LIN {X 0,Y 364.945,Z 184.267,A -85,B 0,C 180,E1 -13027.295,E2 -13027.295} C_VEL
LIN {X 0,Y 368.82,Z 205.112,A -85,B 0,C 180,E1 -13028.057,E2 -13028.057} C_VEL
LIN {X 0,Y 371.05,Z 221.35,A -85,B 0,C 180,E1 -13028.583,E2 -13028.583} C_VEL
LIN {X 0,Y 369.557,Z 293.97,A -85,B 0,C 180,E1 -13030.126,E2 -13030.126} C_VEL
LIN {X 0,Y 368.772,Z 307.522,A -85,B 0,C 180,E1 -13030.626,E2 -13030.626} C_VEL
LIN {X 0,Y 367.784,Z 320.407,A -85,B 0,C 180,E1 -13031.332,E2 -13031.332} C_VEL
LIN {X 0,Y 366.724,Z 331.401,A -85,B 0,C 180,E1 -13032.143,E2 -13032.143} C_VEL
LIN {X 0,Y 365.474,Z 342.946,A -85,B 0,C 180,E1 -13033.234,E2 -13033.234} C_VEL
LIN {X 0,Y 364.338,Z 353.389,A -85,B 0,C 180,E1 -13034.475,E2 -13034.475} C_VEL
LIN {X 0,Y 363.355,Z 361.959,A -85,B 0,C 180,E1 -13035.722,E2 -13035.722} C_VEL
LIN {X 0,Y 362.336,Z 371.27,A -85,B 0,C 180,E1 -13037.395,E2 -13037.395} C_VEL
LIN {X 0,Y 361.44,Z 378.781,A -85,B 0,C 180,E1 -13039.071,E2 -13039.071} C_VEL
LIN {X 0,Y 360.832,Z 385.726,A -85,B 0,C 180,E1 -13041.035,E2 -13041.035} C_VEL
LIN {X 0,Y 360.514,Z 390.327,A -85,B 0,C 180,E1 -13042.72,E2 -13042.72} C_VEL
LIN {X 0,Y 360.354,Z 393.835,A -85,B 0,C 180,E1 -13044.403,E2 -13044.403} C_VEL
LIN {X 0,Y 360.362,Z 395.591,A -85,B 0,C 180,E1 -13045.525,E2 -13045.525} C_VEL
LIN {X 0,Y 360.327,Z 396.936,A -85,B 0,C 180,E1 -13046.645,E2 -13046.645} C_VEL
LIN {X 0,Y 360.353,Z 397.882,A -85,B 0,C 180,E1 -13047.764,E2 -13047.764} C_VEL
LIN {X 0,Y 360.457,Z 398.389,A -85,B 0,C 180,E1 -13048.882,E2 -13048.882} C_VEL
LIN {X 0,Y 360.482,Z 398.479,A -85,B 0,C 180,E1 -13049.999,E2 -13049.999} C_VEL
LIN {X 0,Y 360.459,Z 398.172,A -85,B 0,C 180,E1 -13051.117,E2 -13051.117} C_VEL
LIN {X 0,Y 360.372,Z 397.464,A -85,B 0,C 180,E1 -13052.235,E2 -13052.235} C_VEL
LIN {X 0,Y 360.332,Z 396.308,A -85,B 0,C 180,E1 -13053.354,E2 -13053.354} C_VEL
LIN {X 0,Y 360.343,Z 393.784,A -85,B 0,C 180,E1 -13055.034,E2 -13055.034} C_VEL
LIN {X 0,Y 360.486,Z 390.224,A -85,B 0,C 180,E1 -13056.717,E2 -13056.717} C_VEL
LIN {X 0,Y 360.691,Z 385.523,A -85,B 0,C 180,E1 -13058.402,E2 -13058.402} C_VEL
LIN {X 0,Y 361.168,Z 378.413,A -85,B 0,C 180,E1 -13060.369,E2 -13060.369} C_VEL
LIN {X 0,Y 361.858,Z 370.705,A -85,B 0,C 180,E1 -13062.051,E2 -13062.051} C_VEL
LIN {X 0,Y 362.587,Z 362.799,A -85,B 0,C 180,E1 -13063.449,E2 -13063.449} C_VEL
LIN {X 0,Y 363.508,Z 352.595,A -85,B 0,C 180,E1 -13064.914,E2 -13064.914} C_VEL
LIN {X 0,Y 364.485,Z 342.422,A -85,B 0,C 180,E1 -13066.091,E2 -13066.091} C_VEL
LIN {X 0,Y 365.405,Z 332.091,A -85,B 0,C 180,E1 -13067.056,E2 -13067.056} C_VEL
LIN {X 0,Y 366.377,Z 319.805,A -85,B 0,C 180,E1 -13067.945,E2 -13067.945} C_VEL
LIN {X 0,Y 367.227,Z 306.969,A -85,B 0,C 180,E1 -13068.624,E2 -13068.624} C_VEL
LIN {X 0,Y 367.794,Z 293.504,A -85,B 0,C 180,E1 -13069.1,E2 -13069.1} C_VEL
LIN {X 0,Y 369.081,Z 220.811,A -85,B 0,C 180,E1 -13070.608,E2 -13070.608} C_VEL
LIN {X 0,Y 364.099,Z 185.898,A -85,B 0,C 180,E1 -13071.645,E2 -13071.645} C_VEL
LIN {X 0,Y 365.733,Z 168.533,A -85,B 0,C 180,E1 -13075.422,E2 -13075.422} C_VEL
LIN {X 0,Y 365.024,Z 163.532,A -85,B 0,C 180,E1 -13076.592,E2 -13076.592} C_VEL
LIN {X 0,Y 363.135,Z 153.852,A -85,B 0,C 180,E1 -13078.936,E2 -13078.936} C_VEL
LIN {X 0,Y 361.915,Z 148.405,A -85,B 0,C 180,E1 -13080.323,E2 -13080.323} C_VEL
LIN {X 0,Y 361.856,Z 148.41,A -85,B 0,C 180,E1 -13084.279,E2 -13084.279} C_VEL
LIN {X 0,Y 361.864,Z 148.407,A -85,B 0,C 180,E1 -13087.222,E2 -13087.222} C_VEL
LIN {X 0,Y 361.836,Z 148.41,A -85,B 0,C 180,E1 -13090.755,E2 -13090.755} C_VEL
LIN {X 0,Y 361.817,Z 148.413,A -85,B 0,C 180,E1 -13094.368,E2 -13094.368} C_VEL
LIN {X 0,Y 361.836,Z 148.414,A -85,B 0,C 180,E1 -13097.567,E2 -13097.567} C_VEL
LIN {X 0,Y 361.867,Z 148.406,A -85,B 0,C 180,E1 -13100.973,E2 -13100.973} C_VEL
LIN {X 0,Y 361.873,Z 148.405,A -85,B 0,C 180,E1 -13104.654,E2 -13104.654} C_VEL
LIN {X 0,Y 361.836,Z 148.41,A -85,B 0,C 180,E1 -13108.37,E2 -13108.37} C_VEL
LIN {X 0,Y 361.899,Z 148.403,A -85,B 0,C 180,E1 -13110.955,E2 -13110.955} C_VEL
LIN {X 0,Y 361.954,Z 148.4,A -85,B 0,C 180,E1 -13113.474,E2 -13113.474} C_VEL
LIN {X 0,Y 361.889,Z 148.408,A -85,B 0,C 180,E1 -13117.144,E2 -13117.144} C_VEL
LIN {X 0,Y 361.884,Z 148.405,A -85,B 0,C 180,E1 -13120.722,E2 -13120.722} C_VEL
LIN {X 0,Y 361.942,Z 148.396,A -85,B 0,C 180,E1 -13124.225,E2 -13124.225} C_VEL
LIN {X 0,Y 361.997,Z 148.391,A -85,B 0,C 180,E1 -13126.527,E2 -13126.527} C_VEL
LIN {X 0,Y 362.03,Z 148.386,A -85,B 0,C 180,E1 -13129.937,E2 -13129.937} C_VEL
LIN {X 0,Y 362.159,Z 148.372,A -85,B 0,C 180,E1 -13133.313,E2 -13133.313} C_VEL
LIN {X 0,Y 362.281,Z 148.354,A -85,B 0,C 180,E1 -13137.776,E2 -13137.776} C_VEL
LIN {X 0,Y 362.426,Z 148.336,A -85,B 0,C 180,E1 -13139.999,E2 -13139.999} C_VEL
LIN {X 0,Y 362.28,Z 148.355,A -85,B 0,C 180,E1 -13142.223,E2 -13142.223} C_VEL
LIN {X 0,Y 362.158,Z 148.376,A -85,B 0,C 180,E1 -13146.686,E2 -13146.686} C_VEL
LIN {X 0,Y 362.028,Z 148.387,A -85,B 0,C 180,E1 -13150.061,E2 -13150.061} C_VEL
LIN {X 0,Y 361.994,Z 148.391,A -85,B 0,C 180,E1 -13153.898,E2 -13153.898} C_VEL
LIN {X 0,Y 361.963,Z 148.395,A -85,B 0,C 180,E1 -13157.938,E2 -13157.938} C_VEL
LIN {X 0,Y 361.888,Z 148.404,A -85,B 0,C 180,E1 -13161.652,E2 -13161.652} C_VEL
LIN {X 0,Y 361.924,Z 148.399,A -85,B 0,C 180,E1 -13165.29,E2 -13165.29} C_VEL
LIN {X 0,Y 361.914,Z 148.402,A -85,B 0,C 180,E1 -13167.778,E2 -13167.778} C_VEL
LIN {X 0,Y 361.842,Z 148.409,A -85,B 0,C 180,E1 -13171.285,E2 -13171.285} C_VEL
LIN {X 0,Y 361.85,Z 148.413,A -85,B 0,C 180,E1 -13174.28,E2 -13174.28} C_VEL
LIN {X 0,Y 361.861,Z 148.407,A -85,B 0,C 180,E1 -13177.223,E2 -13177.223} C_VEL
LIN {X 0,Y 361.901,Z 148.402,A -85,B 0,C 180,E1 -13180.768,E2 -13180.768} C_VEL
LIN {X 0,Y 361.929,Z 148.4,A -85,B 0,C 180,E1 -13184.35,E2 -13184.35} C_VEL
LIN {X 0,Y 361.887,Z 148.406,A -85,B 0,C 180,E1 -13187.558,E2 -13187.558} C_VEL
LIN {X 0,Y 361.87,Z 148.406,A -85,B 0,C 180,E1 -13190.972,E2 -13190.972} C_VEL
LIN {X 0,Y 361.869,Z 148.405,A -85,B 0,C 180,E1 -13194.655,E2 -13194.655} C_VEL
LIN {X 0,Y 361.832,Z 148.411,A -85,B 0,C 180,E1 -13198.371,E2 -13198.371} C_VEL
LIN {X 0,Y 361.895,Z 148.403,A -85,B 0,C 180,E1 -13200.955,E2 -13200.955} C_VEL
LIN {X 0,Y 361.949,Z 148.401,A -85,B 0,C 180,E1 -13203.475,E2 -13203.475} C_VEL
LIN {X 0,Y 361.885,Z 148.406,A -85,B 0,C 180,E1 -13207.145,E2 -13207.145} C_VEL
LIN {X 0,Y 361.916,Z 148.4,A -85,B 0,C 180,E1 -13210.725,E2 -13210.725} C_VEL
LIN {X 0,Y 361.942,Z 148.397,A -85,B 0,C 180,E1 -13214.227,E2 -13214.227} C_VEL
LIN {X 0,Y 361.994,Z 148.39,A -85,B 0,C 180,E1 -13216.528,E2 -13216.528} C_VEL
LIN {X 0,Y 362.027,Z 148.386,A -85,B 0,C 180,E1 -13219.939,E2 -13219.939} C_VEL
LIN {X 0,Y 362.147,Z 148.371,A -85,B 0,C 180,E1 -13222.193,E2 -13222.193} C_VEL
LIN {X 0,Y 362.115,Z 148.376,A -85,B 0,C 180,E1 -13224.432,E2 -13224.432} C_VEL
LIN {X 0,Y 362.279,Z 148.355,A -85,B 0,C 180,E1 -13227.777,E2 -13227.777} C_VEL
LIN {X 0,Y 362.425,Z 148.336,A -85,B 0,C 180,E1 -13230.001,E2 -13230.001} C_VEL
LIN {X 0,Y 362.279,Z 148.355,A -85,B 0,C 180,E1 -13232.224,E2 -13232.224} C_VEL
LIN {X 0,Y 362.17,Z 148.373,A -85,B 0,C 180,E1 -13236.687,E2 -13236.687} C_VEL
LIN {X 0,Y 362.071,Z 148.385,A -85,B 0,C 180,E1 -13238.934,E2 -13238.934} C_VEL
LIN {X 0,Y 361.955,Z 148.397,A -85,B 0,C 180,E1 -13242.333,E2 -13242.333} C_VEL
LIN {X 0,Y 361.988,Z 148.454,A -85,B 0,C 180,E1 -13244.692,E2 -13244.692} C_VEL
LIN {X 0,Y 363.275,Z 154.799,A -85,B 0,C 180,E1 -13246.4,E2 -13246.4} C_VEL
LIN {X 0,Y 367.605,Z 168.073,A -85,B 0,C 180,E1 -13246.933,E2 -13246.933} C_VEL
LIN {X 0,Y 369.738,Z 179.441,A -85,B 0,C 180,E1 -13247.294,E2 -13247.294} C_VEL
LIN {X 0,Y 368.028,Z 262.471,A -85,B 0,C 180,E1 -13249.017,E2 -13249.017} C_VEL
LIN {X 0,Y 367.494,Z 276.574,A -85,B 0,C 180,E1 -13249.553,E2 -13249.553} C_VEL
LIN {X 0,Y 366.864,Z 289.461,A -85,B 0,C 180,E1 -13250.29,E2 -13250.29} C_VEL
LIN {X 0,Y 366.118,Z 301.585,A -85,B 0,C 180,E1 -13251.229,E2 -13251.229} C_VEL
LIN {X 0,Y 365.138,Z 312.893,A -85,B 0,C 180,E1 -13252.343,E2 -13252.343} C_VEL
LIN {X 0,Y 364.402,Z 320.864,A -85,B 0,C 180,E1 -13253.312,E2 -13253.312} C_VEL
LIN {X 0,Y 363.351,Z 325.335,A -85,B 0,C 180,E1 -13253.898,E2 -13253.898} C_VEL
LIN {X 0,Y 359.883,Z 332.258,A -85,B 0,C 180,E1 -13254.882,E2 -13254.882} C_VEL
LIN {X 0,Y 356.434,Z 338.658,A -85,B 0,C 180,E1 -13255.967,E2 -13255.967} C_VEL
LIN {X 0,Y 355.427,Z 342.237,A -85,B 0,C 180,E1 -13256.704,E2 -13256.704} C_VEL
LIN {X 0,Y 354.725,Z 349.044,A -85,B 0,C 180,E1 -13258.393,E2 -13258.393} C_VEL
LIN {X 0,Y 354.107,Z 355.412,A -85,B 0,C 180,E1 -13260.405,E2 -13260.405} C_VEL
LIN {X 0,Y 353.805,Z 358.939,A -85,B 0,C 180,E1 -13261.856,E2 -13261.856} C_VEL
LIN {X 0,Y 353.427,Z 362.572,A -85,B 0,C 180,E1 -13263.835,E2 -13263.835} C_VEL
LIN {X 0,Y 353.208,Z 364.417,A -85,B 0,C 180,E1 -13265.334,E2 -13265.334} C_VEL
LIN {X 0,Y 353.107,Z 365.757,A -85,B 0,C 180,E1 -13267.239,E2 -13267.239} C_VEL
LIN {X 0,Y 353.161,Z 365.882,A -85,B 0,C 180,E1 -13269.555,E2 -13269.555} C_VEL
LIN {X 0,Y 353.304,Z 365.095,A -85,B 0,C 180,E1 -13271.03,E2 -13271.03} C_VEL
LIN {X 0,Y 353.678,Z 362.529,A -85,B 0,C 180,E1 -13273.305,E2 -13273.305} C_VEL
LIN {X 0,Y 354.088,Z 359.677,A -85,B 0,C 180,E1 -13274.926,E2 -13274.926} C_VEL
LIN {X 0,Y 354.526,Z 355.892,A -85,B 0,C 180,E1 -13276.547,E2 -13276.547} C_VEL
LIN {X 0,Y 355.219,Z 351.09,A -85,B 0,C 180,E1 -13278.152,E2 -13278.152} C_VEL
LIN {X 0,Y 356.131,Z 343.991,A -85,B 0,C 180,E1 -13280.021,E2 -13280.021} C_VEL
LIN {X 0,Y 357.199,Z 335.856,A -85,B 0,C 180,E1 -13281.723,E2 -13281.723} C_VEL
LIN {X 0,Y 358.174,Z 328.163,A -85,B 0,C 180,E1 -13283.033,E2 -13283.033} C_VEL
LIN {X 0,Y 359.227,Z 319.028,A -85,B 0,C 180,E1 -13284.323,E2 -13284.323} C_VEL
LIN {X 0,Y 360.503,Z 307.89,A -85,B 0,C 180,E1 -13285.574,E2 -13285.574} C_VEL
LIN {X 0,Y 361.665,Z 295.388,A -85,B 0,C 180,E1 -13286.679,E2 -13286.679} C_VEL
LIN {X 0,Y 362.559,Z 282.676,A -85,B 0,C 180,E1 -13287.515,E2 -13287.515} C_VEL
LIN {X 0,Y 363.168,Z 269.986,A -85,B 0,C 180,E1 -13288.113,E2 -13288.113} C_VEL
LIN {X 0,Y 363.672,Z 257.174,A -85,B 0,C 180,E1 -13288.487,E2 -13288.487} C_VEL
LIN {X 0,Y 365.352,Z 180.512,A -85,B 0,C 180,E1 -13290.133,E2 -13290.133} C_VEL
LIN {X 0,Y 363.652,Z 173.572,A -85,B 0,C 180,E1 -13290.423,E2 -13290.423} C_VEL
LIN {X 0,Y 357.382,Z 158.56,A -85,B 0,C 180,E1 -13291.278,E2 -13291.278} C_VEL
LIN {X 0,Y 356.459,Z 156.273,A -85,B 0,C 180,E1 -13291.438,E2 -13291.438} C_VEL
LIN {X 0,Y 354.923,Z 149.279,A -85,B 0,C 180,E1 -13293.543,E2 -13293.543} C_VEL
LIN {X 0,Y 354.829,Z 149.292,A -85,B 0,C 180,E1 -13296.664,E2 -13296.664} C_VEL
LIN {X 0,Y 354.847,Z 149.285,A -85,B 0,C 180,E1 -13300.325,E2 -13300.325} C_VEL
LIN {X 0,Y 354.89,Z 149.279,A -85,B 0,C 180,E1 -13303.905,E2 -13303.905} C_VEL
LIN {X 0,Y 354.925,Z 149.278,A -85,B 0,C 180,E1 -13307.42,E2 -13307.42} C_VEL
LIN {X 0,Y 354.998,Z 149.271,A -85,B 0,C 180,E1 -13310.888,E2 -13310.888} C_VEL
LIN {X 0,Y 355.07,Z 149.261,A -85,B 0,C 180,E1 -13314.321,E2 -13314.321} C_VEL
LIN {X 0,Y 355.232,Z 149.237,A -85,B 0,C 180,E1 -13317.733,E2 -13317.733} C_VEL
LIN {X 0,Y 355.151,Z 149.245,A -85,B 0,C 180,E1 -13321.135,E2 -13321.135} C_VEL
LIN {X 0,Y 355.224,Z 149.231,A -85,B 0,C 180,E1 -13322.268,E2 -13322.268} C_VEL
LIN {X 0,Y 355.094,Z 149.242,A -85,B 0,C 180,E1 -13326.821,E2 -13326.821} C_VEL
LIN {X 0,Y 354.954,Z 149.262,A -85,B 0,C 180,E1 -13330.265,E2 -13330.265} C_VEL
LIN {X 0,Y 354.897,Z 149.273,A -85,B 0,C 180,E1 -13333.986,E2 -13333.986} C_VEL
LIN {X 0,Y 354.838,Z 149.281,A -85,B 0,C 180,E1 -13338.064,E2 -13338.064} C_VEL
LIN {X 0,Y 354.791,Z 149.289,A -85,B 0,C 180,E1 -13342.11,E2 -13342.11} C_VEL
LIN {X 0,Y 354.799,Z 149.289,A -85,B 0,C 180,E1 -13345.836,E2 -13345.836} C_VEL
LIN {X 0,Y 354.798,Z 149.289,A -85,B 0,C 180,E1 -13349.684,E2 -13349.684} C_VEL
LIN {X 0,Y 354.789,Z 149.286,A -85,B 0,C 180,E1 -13352.334,E2 -13352.334} C_VEL
LIN {X 0,Y 354.826,Z 149.284,A -85,B 0,C 180,E1 -13355.699,E2 -13355.699} C_VEL
LIN {X 0,Y 354.773,Z 149.293,A -85,B 0,C 180,E1 -13359.412,E2 -13359.412} C_VEL
LIN {X 0,Y 354.789,Z 149.294,A -85,B 0,C 180,E1 -13362.866,E2 -13362.866} C_VEL
LIN {X 0,Y 354.77,Z 149.296,A -85,B 0,C 180,E1 -13366.103,E2 -13366.103} C_VEL
LIN {X 0,Y 354.771,Z 149.296,A -85,B 0,C 180,E1 -13369.176,E2 -13369.176} C_VEL
LIN {X 0,Y 354.805,Z 149.29,A -85,B 0,C 180,E1 -13372.404,E2 -13372.404} C_VEL
LIN {X 0,Y 354.817,Z 149.289,A -85,B 0,C 180,E1 -13374.941,E2 -13374.941} C_VEL
LIN {X 0,Y 354.83,Z 149.428,A -85,B 0,C 180,E1 -13378.247,E2 -13378.247} C_VEL
LIN {X 0,Y 357.476,Z 160.388,A -85,B 0,C 180,E1 -13381.205,E2 -13381.205} C_VEL
LIN {X 0,Y 359.478,Z 170.683,A -85,B 0,C 180,E1 -13383.815,E2 -13383.815} C_VEL
LIN {X 0,Y 358.423,Z 182.015,A -85,B 0,C 180,E1 -13386.359,E2 -13386.359} C_VEL
LIN {X 0,Y 358.244,Z 184.062,A -85,B 0,C 180,E1 -13386.774,E2 -13386.774} C_VEL
LIN {X 0,Y 362.351,Z 205.998,A -85,B 0,C 180,E1 -13387.608,E2 -13387.608} C_VEL
LIN {X 0,Y 364.57,Z 222.715,A -85,B 0,C 180,E1 -13388.158,E2 -13388.158} C_VEL
LIN {X 0,Y 362.964,Z 294.03,A -85,B 0,C 180,E1 -13389.713,E2 -13389.713} C_VEL
LIN {X 0,Y 362.162,Z 307.409,A -85,B 0,C 180,E1 -13390.221,E2 -13390.221} C_VEL
LIN {X 0,Y 361.191,Z 319.691,A -85,B 0,C 180,E1 -13390.904,E2 -13390.904} C_VEL
LIN {X 0,Y 360.158,Z 329.964,A -85,B 0,C 180,E1 -13391.659,E2 -13391.659} C_VEL
LIN {X 0,Y 358.83,Z 341.724,A -85,B 0,C 180,E1 -13392.768,E2 -13392.768} C_VEL
LIN {X 0,Y 357.618,Z 352.32,A -85,B 0,C 180,E1 -13394.029,E2 -13394.029} C_VEL
LIN {X 0,Y 356.474,Z 361.906,A -85,B 0,C 180,E1 -13395.441,E2 -13395.441} C_VEL
LIN {X 0,Y 355.371,Z 371.156,A -85,B 0,C 180,E1 -13397.144,E2 -13397.144} C_VEL
LIN {X 0,Y 354.417,Z 378.632,A -85,B 0,C 180,E1 -13398.852,E2 -13398.852} C_VEL
LIN {X 0,Y 353.943,Z 383.723,A -85,B 0,C 180,E1 -13400.283,E2 -13400.283} C_VEL
LIN {X 0,Y 353.545,Z 388.683,A -85,B 0,C 180,E1 -13402.001,E2 -13402.001} C_VEL
LIN {X 0,Y 353.28,Z 393.23,A -85,B 0,C 180,E1 -13404.091,E2 -13404.091} C_VEL
LIN {X 0,Y 353.272,Z 395.314,A -85,B 0,C 180,E1 -13405.435,E2 -13405.435} C_VEL
LIN {X 0,Y 353.246,Z 396.649,A -85,B 0,C 180,E1 -13406.578,E2 -13406.578} C_VEL
LIN {X 0,Y 353.255,Z 397.58,A -85,B 0,C 180,E1 -13407.719,E2 -13407.719} C_VEL
LIN {X 0,Y 353.358,Z 398.068,A -85,B 0,C 180,E1 -13408.86,E2 -13408.86} C_VEL
LIN {X 0,Y 353.401,Z 398.148,A -85,B 0,C 180,E1 -13409.999,E2 -13409.999} C_VEL
LIN {X 0,Y 353.362,Z 397.828,A -85,B 0,C 180,E1 -13411.139,E2 -13411.139} C_VEL
LIN {X 0,Y 353.274,Z 397.105,A -85,B 0,C 180,E1 -13412.28,E2 -13412.28} C_VEL
LIN {X 0,Y 353.252,Z 395.927,A -85,B 0,C 180,E1 -13413.421,E2 -13413.421} C_VEL
LIN {X 0,Y 353.248,Z 393.375,A -85,B 0,C 180,E1 -13415.136,E2 -13415.136} C_VEL
LIN {X 0,Y 353.396,Z 389.784,A -85,B 0,C 180,E1 -13416.852,E2 -13416.852} C_VEL
LIN {X 0,Y 353.637,Z 385.05,A -85,B 0,C 180,E1 -13418.571,E2 -13418.571} C_VEL
LIN {X 0,Y 354.133,Z 377.902,A -85,B 0,C 180,E1 -13420.577,E2 -13420.577} C_VEL
LIN {X 0,Y 354.876,Z 370.14,A -85,B 0,C 180,E1 -13422.291,E2 -13422.291} C_VEL
LIN {X 0,Y 355.86,Z 360.447,A -85,B 0,C 180,E1 -13423.988,E2 -13423.988} C_VEL
LIN {X 0,Y 356.761,Z 350.717,A -85,B 0,C 180,E1 -13425.364,E2 -13425.364} C_VEL
LIN {X 0,Y 357.712,Z 340.295,A -85,B 0,C 180,E1 -13426.551,E2 -13426.551} C_VEL
LIN {X 0,Y 358.88,Z 327.697,A -85,B 0,C 180,E1 -13427.67,E2 -13427.67} C_VEL
LIN {X 0,Y 359.833,Z 315.294,A -85,B 0,C 180,E1 -13428.504,E2 -13428.504} C_VEL
LIN {X 0,Y 360.62,Z 302.184,A -85,B 0,C 180,E1 -13429.126,E2 -13429.126} C_VEL
LIN {X 0,Y 361.143,Z 288.314,A -85,B 0,C 180,E1 -13429.54,E2 -13429.54} C_VEL
LIN {X 0,Y 362.285,Z 221.025,A -85,B 0,C 180,E1 -13430.954,E2 -13430.954} C_VEL
LIN {X 0,Y 357.212,Z 185.502,A -85,B 0,C 180,E1 -13432.048,E2 -13432.048} C_VEL
LIN {X 0,Y 358.761,Z 169.82,A -85,B 0,C 180,E1 -13435.529,E2 -13435.529} C_VEL
LIN {X 0,Y 358.231,Z 165.702,A -85,B 0,C 180,E1 -13436.509,E2 -13436.509} C_VEL
LIN {X 0,Y 356.025,Z 154.607,A -85,B 0,C 180,E1 -13439.246,E2 -13439.246} C_VEL
LIN {X 0,Y 354.837,Z 149.284,A -85,B 0,C 180,E1 -13440.664,E2 -13440.664} C_VEL
LIN {X 0,Y 354.807,Z 149.289,A -85,B 0,C 180,E1 -13443.701,E2 -13443.701} C_VEL
LIN {X 0,Y 354.799,Z 149.288,A -85,B 0,C 180,E1 -13446.459,E2 -13446.459} C_VEL
LIN {X 0,Y 354.824,Z 149.285,A -85,B 0,C 180,E1 -13449.423,E2 -13449.423} C_VEL
LIN {X 0,Y 354.788,Z 149.288,A -85,B 0,C 180,E1 -13452.866,E2 -13452.866} C_VEL
LIN {X 0,Y 354.767,Z 149.293,A -85,B 0,C 180,E1 -13456.103,E2 -13456.103} C_VEL
LIN {X 0,Y 354.787,Z 149.289,A -85,B 0,C 180,E1 -13459.178,E2 -13459.178} C_VEL
LIN {X 0,Y 354.806,Z 149.286,A -85,B 0,C 180,E1 -13462.402,E2 -13462.402} C_VEL
LIN {X 0,Y 354.811,Z 149.286,A -85,B 0,C 180,E1 -13464.94,E2 -13464.94} C_VEL
LIN {X 0,Y 354.792,Z 149.287,A -85,B 0,C 180,E1 -13468.404,E2 -13468.404} C_VEL
LIN {X 0,Y 354.85,Z 149.284,A -85,B 0,C 180,E1 -13471.618,E2 -13471.618} C_VEL
LIN {X 0,Y 354.898,Z 149.274,A -85,B 0,C 180,E1 -13474.172,E2 -13474.172} C_VEL
LIN {X 0,Y 354.834,Z 149.283,A -85,B 0,C 180,E1 -13477.893,E2 -13477.893} C_VEL
LIN {X 0,Y 354.888,Z 149.276,A -85,B 0,C 180,E1 -13481.907,E2 -13481.907} C_VEL
LIN {X 0,Y 354.941,Z 149.269,A -85,B 0,C 180,E1 -13485.98,E2 -13485.98} C_VEL
LIN {X 0,Y 354.976,Z 149.265,A -85,B 0,C 180,E1 -13489.735,E2 -13489.735} C_VEL
LIN {X 0,Y 355.123,Z 149.25,A -85,B 0,C 180,E1 -13493.18,E2 -13493.18} C_VEL
LIN {X 0,Y 355.244,Z 149.231,A -85,B 0,C 180,E1 -13497.732,E2 -13497.732} C_VEL
LIN {X 0,Y 355.395,Z 149.212,A -85,B 0,C 180,E1 -13499.999,E2 -13499.999} C_VEL
LIN {X 0,Y 355.243,Z 149.232,A -85,B 0,C 180,E1 -13502.267,E2 -13502.267} C_VEL
LIN {X 0,Y 355.122,Z 149.251,A -85,B 0,C 180,E1 -13506.819,E2 -13506.819} C_VEL
LIN {X 0,Y 354.975,Z 149.267,A -85,B 0,C 180,E1 -13510.264,E2 -13510.264} C_VEL
LIN {X 0,Y 354.939,Z 149.27,A -85,B 0,C 180,E1 -13514.018,E2 -13514.018} C_VEL
LIN {X 0,Y 354.919,Z 149.274,A -85,B 0,C 180,E1 -13518.108,E2 -13518.108} C_VEL
LIN {X 0,Y 354.831,Z 149.286,A -85,B 0,C 180,E1 -13522.106,E2 -13522.106} C_VEL
LIN {X 0,Y 354.895,Z 149.276,A -85,B 0,C 180,E1 -13525.827,E2 -13525.827} C_VEL
LIN {X 0,Y 354.849,Z 149.281,A -85,B 0,C 180,E1 -13529.678,E2 -13529.678} C_VEL
LIN {X 0,Y 354.801,Z 149.288,A -85,B 0,C 180,E1 -13533.702,E2 -13533.702} C_VEL
LIN {X 0,Y 354.795,Z 149.289,A -85,B 0,C 180,E1 -13536.459,E2 -13536.459} C_VEL
LIN {X 0,Y 354.819,Z 149.285,A -85,B 0,C 180,E1 -13539.423,E2 -13539.423} C_VEL
LIN {X 0,Y 354.84,Z 149.281,A -85,B 0,C 180,E1 -13542.877,E2 -13542.877} C_VEL
LIN {X 0,Y 354.863,Z 149.282,A -85,B 0,C 180,E1 -13546.119,E2 -13546.119} C_VEL
LIN {X 0,Y 354.852,Z 149.28,A -85,B 0,C 180,E1 -13549.189,E2 -13549.189} C_VEL
LIN {X 0,Y 354.804,Z 149.286,A -85,B 0,C 180,E1 -13552.402,E2 -13552.402} C_VEL
LIN {X 0,Y 354.807,Z 149.286,A -85,B 0,C 180,E1 -13554.941,E2 -13554.941} C_VEL
LIN {X 0,Y 354.788,Z 149.288,A -85,B 0,C 180,E1 -13558.405,E2 -13558.405} C_VEL
LIN {X 0,Y 354.846,Z 149.286,A -85,B 0,C 180,E1 -13561.619,E2 -13561.619} C_VEL
LIN {X 0,Y 354.894,Z 149.275,A -85,B 0,C 180,E1 -13564.173,E2 -13564.173} C_VEL
LIN {X 0,Y 354.83,Z 149.284,A -85,B 0,C 180,E1 -13567.894,E2 -13567.894} C_VEL
LIN {X 0,Y 354.918,Z 149.273,A -85,B 0,C 180,E1 -13571.892,E2 -13571.892} C_VEL
LIN {X 0,Y 354.938,Z 149.27,A -85,B 0,C 180,E1 -13575.982,E2 -13575.982} C_VEL
LIN {X 0,Y 354.974,Z 149.266,A -85,B 0,C 180,E1 -13579.736,E2 -13579.736} C_VEL
LIN {X 0,Y 355.11,Z 149.248,A -85,B 0,C 180,E1 -13582.037,E2 -13582.037} C_VEL
LIN {X 0,Y 355.089,Z 149.25,A -85,B 0,C 180,E1 -13584.321,E2 -13584.321} C_VEL
LIN {X 0,Y 355.242,Z 149.232,A -85,B 0,C 180,E1 -13587.733,E2 -13587.733} C_VEL
LIN {X 0,Y 355.394,Z 149.212,A -85,B 0,C 180,E1 -13590.001,E2 -13590.001} C_VEL
LIN {X 0,Y 355.243,Z 149.232,A -85,B 0,C 180,E1 -13592.268,E2 -13592.268} C_VEL
LIN {X 0,Y 355.136,Z 149.25,A -85,B 0,C 180,E1 -13596.82,E2 -13596.82} C_VEL
LIN {X 0,Y 355.012,Z 149.263,A -85,B 0,C 180,E1 -13599.113,E2 -13599.113} C_VEL
LIN {X 0,Y 354.917,Z 149.276,A -85,B 0,C 180,E1 -13602.582,E2 -13602.582} C_VEL
LIN {X 0,Y 354.985,Z 149.42,A -85,B 0,C 180,E1 -13604.444,E2 -13604.444} C_VEL
LIN {X 0,Y 356.129,Z 155.025,A -85,B 0,C 180,E1 -13606.002,E2 -13606.002} C_VEL
LIN {X 0,Y 361.159,Z 170.41,A -85,B 0,C 180,E1 -13606.632,E2 -13606.632} C_VEL
LIN {X 0,Y 363.005,Z 179.959,A -85,B 0,C 180,E1 -13606.944,E2 -13606.944} C_VEL
LIN {X 0,Y 361.243,Z 262.464,A -85,B 0,C 180,E1 -13608.688,E2 -13608.688} C_VEL
LIN {X 0,Y 360.689,Z 275.9,A -85,B 0,C 180,E1 -13609.197,E2 -13609.197} C_VEL
LIN {X 0,Y 360.08,Z 288.98,A -85,B 0,C 180,E1 -13609.939,E2 -13609.939} C_VEL
LIN {X 0,Y 359.392,Z 299.755,A -85,B 0,C 180,E1 -13610.76,E2 -13610.76} C_VEL
LIN {X 0,Y 358.395,Z 311.289,A -85,B 0,C 180,E1 -13611.876,E2 -13611.876} C_VEL
LIN {X 0,Y 357.426,Z 321.84,A -85,B 0,C 180,E1 -13613.158,E2 -13613.158} C_VEL
LIN {X 0,Y 356.474,Z 331.699,A -85,B 0,C 180,E1 -13614.66,E2 -13614.66} C_VEL
LIN {X 0,Y 355.561,Z 340.886,A -85,B 0,C 180,E1 -13616.407,E2 -13616.407} C_VEL
LIN {X 0,Y 355.427,Z 342.237,A -85,B 0,C 180,E1 -13616.704,E2 -13616.704} C_VEL
LIN {X 0,Y 354.437,Z 345.626,A -85,B 0,C 180,E1 -13617.47,E2 -13617.47} C_VEL
LIN {X 0,Y 351.078,Z 350.689,A -85,B 0,C 180,E1 -13618.744,E2 -13618.744} C_VEL
LIN {X 0,Y 347.778,Z 355.111,A -85,B 0,C 180,E1 -13620.102,E2 -13620.102} C_VEL
LIN {X 0,Y 346.9,Z 357.443,A -85,B 0,C 180,E1 -13620.985,E2 -13620.985} C_VEL
LIN {X 0,Y 346.463,Z 361.961,A -85,B 0,C 180,E1 -13623.21,E2 -13623.21} C_VEL
LIN {X 0,Y 346.19,Z 364.001,A -85,B 0,C 180,E1 -13624.642,E2 -13624.642} C_VEL
LIN {X 0,Y 346.048,Z 365.396,A -85,B 0,C 180,E1 -13626.085,E2 -13626.085} C_VEL
LIN {X 0,Y 346.013,Z 366.225,A -85,B 0,C 180,E1 -13627.615,E2 -13627.615} C_VEL
LIN {X 0,Y 346.093,Z 366.262,A -85,B 0,C 180,E1 -13629.499,E2 -13629.499} C_VEL
LIN {X 0,Y 346.274,Z 365.294,A -85,B 0,C 180,E1 -13631.328,E2 -13631.328} C_VEL
LIN {X 0,Y 346.667,Z 362.694,A -85,B 0,C 180,E1 -13633.574,E2 -13633.574} C_VEL
LIN {X 0,Y 347.07,Z 359.975,A -85,B 0,C 180,E1 -13635.133,E2 -13635.133} C_VEL
LIN {X 0,Y 347.666,Z 355.313,A -85,B 0,C 180,E1 -13637.102,E2 -13637.102} C_VEL
LIN {X 0,Y 348.55,Z 349.068,A -85,B 0,C 180,E1 -13639.095,E2 -13639.095} C_VEL
LIN {X 0,Y 349.493,Z 342.626,A -85,B 0,C 180,E1 -13640.712,E2 -13640.712} C_VEL
LIN {X 0,Y 350.652,Z 333.977,A -85,B 0,C 180,E1 -13642.455,E2 -13642.455} C_VEL
LIN {X 0,Y 351.869,Z 325.088,A -85,B 0,C 180,E1 -13643.9,E2 -13643.9} C_VEL
LIN {X 0,Y 352.96,Z 315.862,A -85,B 0,C 180,E1 -13645.13,E2 -13645.13} C_VEL
LIN {X 0,Y 354.207,Z 305.429,A -85,B 0,C 180,E1 -13646.251,E2 -13646.251} C_VEL
LIN {X 0,Y 355.223,Z 294.222,A -85,B 0,C 180,E1 -13647.208,E2 -13647.208} C_VEL
LIN {X 0,Y 356.125,Z 281.01,A -85,B 0,C 180,E1 -13648.06,E2 -13648.06} C_VEL
LIN {X 0,Y 356.732,Z 267.761,A -85,B 0,C 180,E1 -13648.653,E2 -13648.653} C_VEL
LIN {X 0,Y 357.306,Z 250.069,A -85,B 0,C 180,E1 -13649.1,E2 -13649.1} C_VEL
LIN {X 0,Y 359.048,Z 182.296,A -85,B 0,C 180,E1 -13650.57,E2 -13650.57} C_VEL
LIN {X 0,Y 357.661,Z 176.495,A -85,B 0,C 180,E1 -13650.82,E2 -13650.82} C_VEL
LIN {X 0,Y 351.543,Z 161.77,A -85,B 0,C 180,E1 -13651.687,E2 -13651.687} C_VEL
LIN {X 0,Y 349.372,Z 156.652,A -85,B 0,C 180,E1 -13652.034,E2 -13652.034} C_VEL
LIN {X 0,Y 347.869,Z 150.159,A -85,B 0,C 180,E1 -13654.015,E2 -13654.015} C_VEL
LIN {X 0,Y 347.765,Z 150.17,A -85,B 0,C 180,E1 -13657.421,E2 -13657.421} C_VEL
LIN {X 0,Y 347.801,Z 150.163,A -85,B 0,C 180,E1 -13661.137,E2 -13661.137} C_VEL
LIN {X 0,Y 347.868,Z 150.154,A -85,B 0,C 180,E1 -13664.774,E2 -13664.774} C_VEL
LIN {X 0,Y 347.888,Z 150.157,A -85,B 0,C 180,E1 -13668.346,E2 -13668.346} C_VEL
LIN {X 0,Y 348.002,Z 150.139,A -85,B 0,C 180,E1 -13671.874,E2 -13671.874} C_VEL
LIN {X 0,Y 348.044,Z 150.136,A -85,B 0,C 180,E1 -13674.206,E2 -13674.206} C_VEL
LIN {X 0,Y 348.193,Z 150.114,A -85,B 0,C 180,E1 -13677.687,E2 -13677.687} C_VEL
LIN {X 0,Y 348.122,Z 150.121,A -85,B 0,C 180,E1 -13681.157,E2 -13681.157} C_VEL
LIN {X 0,Y 348.185,Z 150.107,A -85,B 0,C 180,E1 -13682.314,E2 -13682.314} C_VEL
LIN {X 0,Y 348.061,Z 150.117,A -85,B 0,C 180,E1 -13686.959,E2 -13686.959} C_VEL
LIN {X 0,Y 347.893,Z 150.14,A -85,B 0,C 180,E1 -13690.476,E2 -13690.476} C_VEL
LIN {X 0,Y 347.857,Z 150.148,A -85,B 0,C 180,E1 -13694.119,E2 -13694.119} C_VEL
LIN {X 0,Y 347.791,Z 150.158,A -85,B 0,C 180,E1 -13698.238,E2 -13698.238} C_VEL
LIN {X 0,Y 347.748,Z 150.17,A -85,B 0,C 180,E1 -13701.616,E2 -13701.616} C_VEL
LIN {X 0,Y 347.738,Z 150.167,A -85,B 0,C 180,E1 -13705.115,E2 -13705.115} C_VEL
LIN {X 0,Y 347.729,Z 150.163,A -85,B 0,C 180,E1 -13707.702,E2 -13707.702} C_VEL
LIN {X 0,Y 347.74,Z 150.168,A -85,B 0,C 180,E1 -13710.349,E2 -13710.349} C_VEL
LIN {X 0,Y 347.754,Z 150.165,A -85,B 0,C 180,E1 -13714.044,E2 -13714.044} C_VEL
LIN {X 0,Y 347.762,Z 150.164,A -85,B 0,C 180,E1 -13717.322,E2 -13717.322} C_VEL
LIN {X 0,Y 347.746,Z 150.166,A -85,B 0,C 180,E1 -13721.601,E2 -13721.601} C_VEL
LIN {X 0,Y 347.708,Z 150.178,A -85,B 0,C 180,E1 -13725.027,E2 -13725.027} C_VEL
LIN {X 0,Y 347.746,Z 150.171,A -85,B 0,C 180,E1 -13728.399,E2 -13728.399} C_VEL
LIN {X 0,Y 347.761,Z 150.167,A -85,B 0,C 180,E1 -13732.678,E2 -13732.678} C_VEL
LIN {X 0,Y 347.753,Z 150.172,A -85,B 0,C 180,E1 -13735.956,E2 -13735.956} C_VEL
LIN {X 0,Y 347.77,Z 150.255,A -85,B 0,C 180,E1 -13737.718,E2 -13737.718} C_VEL
LIN {X 0,Y 350.597,Z 161.753,A -85,B 0,C 180,E1 -13740.914,E2 -13740.914} C_VEL
LIN {X 0,Y 352.452,Z 170.96,A -85,B 0,C 180,E1 -13743.316,E2 -13743.316} C_VEL
LIN {X 0,Y 352.63,Z 173.733,A -85,B 0,C 180,E1 -13743.993,E2 -13743.993} C_VEL
LIN {X 0,Y 351.535,Z 183.552,A -85,B 0,C 180,E1 -13746.22,E2 -13746.22} C_VEL
LIN {X 0,Y 355.944,Z 207.012,A -85,B 0,C 180,E1 -13747.148,E2 -13747.148} C_VEL
LIN {X 0,Y 358.11,Z 222.742,A -85,B 0,C 180,E1 -13747.686,E2 -13747.686} C_VEL
LIN {X 0,Y 356.451,Z 293.276,A -85,B 0,C 180,E1 -13749.25,E2 -13749.25} C_VEL
LIN {X 0,Y 355.589,Z 307.517,A -85,B 0,C 180,E1 -13749.802,E2 -13749.802} C_VEL
LIN {X 0,Y 354.513,Z 320.139,A -85,B 0,C 180,E1 -13750.53,E2 -13750.53} C_VEL
LIN {X 0,Y 353.453,Z 330.234,A -85,B 0,C 180,E1 -13751.298,E2 -13751.298} C_VEL
LIN {X 0,Y 352.076,Z 341.845,A -85,B 0,C 180,E1 -13752.426,E2 -13752.426} C_VEL
LIN {X 0,Y 350.767,Z 352.343,A -85,B 0,C 180,E1 -13753.709,E2 -13753.709} C_VEL
LIN {X 0,Y 349.6,Z 361.843,A -85,B 0,C 180,E1 -13755.148,E2 -13755.148} C_VEL
LIN {X 0,Y 348.429,Z 371.045,A -85,B 0,C 180,E1 -13756.884,E2 -13756.884} C_VEL
LIN {X 0,Y 347.418,Z 378.484,A -85,B 0,C 180,E1 -13758.624,E2 -13758.624} C_VEL
LIN {X 0,Y 346.913,Z 383.543,A -85,B 0,C 180,E1 -13760.084,E2 -13760.084} C_VEL
LIN {X 0,Y 346.497,Z 388.473,A -85,B 0,C 180,E1 -13761.837,E2 -13761.837} C_VEL
LIN {X 0,Y 346.227,Z 392.274,A -85,B 0,C 180,E1 -13763.59,E2 -13763.59} C_VEL
LIN {X 0,Y 346.169,Z 395.047,A -85,B 0,C 180,E1 -13765.341,E2 -13765.341} C_VEL
LIN {X 0,Y 346.167,Z 396.369,A -85,B 0,C 180,E1 -13766.507,E2 -13766.507} C_VEL
LIN {X 0,Y 346.16,Z 397.28,A -85,B 0,C 180,E1 -13767.672,E2 -13767.672} C_VEL
LIN {X 0,Y 346.26,Z 397.747,A -85,B 0,C 180,E1 -13768.836,E2 -13768.836} C_VEL
LIN {X 0,Y 346.321,Z 397.815,A -85,B 0,C 180,E1 -13769.999,E2 -13769.999} C_VEL
LIN {X 0,Y 346.264,Z 397.482,A -85,B 0,C 180,E1 -13771.162,E2 -13771.162} C_VEL
LIN {X 0,Y 346.178,Z 396.739,A -85,B 0,C 180,E1 -13772.326,E2 -13772.326} C_VEL
LIN {X 0,Y 346.174,Z 395.542,A -85,B 0,C 180,E1 -13773.491,E2 -13773.491} C_VEL
LIN {X 0,Y 346.167,Z 392.584,A -85,B 0,C 180,E1 -13775.444,E2 -13775.444} C_VEL
LIN {X 0,Y 346.379,Z 387.887,A -85,B 0,C 180,E1 -13777.578,E2 -13777.578} C_VEL
LIN {X 0,Y 346.783,Z 381.709,A -85,B 0,C 180,E1 -13779.624,E2 -13779.624} C_VEL
LIN {X 0,Y 347.295,Z 374.931,A -85,B 0,C 180,E1 -13781.379,E2 -13781.379} C_VEL
LIN {X 0,Y 348.24,Z 366.525,A -85,B 0,C 180,E1 -13783.122,E2 -13783.122} C_VEL
LIN {X 0,Y 349.126,Z 357.357,A -85,B 0,C 180,E1 -13784.647,E2 -13784.647} C_VEL
LIN {X 0,Y 350.063,Z 347.132,A -85,B 0,C 180,E1 -13786.024,E2 -13786.024} C_VEL
LIN {X 0,Y 351.172,Z 336.535,A -85,B 0,C 180,E1 -13787.168,E2 -13787.168} C_VEL
LIN {X 0,Y 352.206,Z 324.785,A -85,B 0,C 180,E1 -13788.166,E2 -13788.166} C_VEL
LIN {X 0,Y 353.268,Z 311.353,A -85,B 0,C 180,E1 -13789.011,E2 -13789.011} C_VEL
LIN {X 0,Y 354.003,Z 298.541,A -85,B 0,C 180,E1 -13789.573,E2 -13789.573} C_VEL
LIN {X 0,Y 354.505,Z 282.21,A -85,B 0,C 180,E1 -13789.99,E2 -13789.99} C_VEL
LIN {X 0,Y 355.48,Z 221.356,A -85,B 0,C 180,E1 -13791.301,E2 -13791.301} C_VEL
LIN {X 0,Y 350.331,Z 185.229,A -85,B 0,C 180,E1 -13792.44,E2 -13792.44} C_VEL
LIN {X 0,Y 351.818,Z 170.391,A -85,B 0,C 180,E1 -13795.801,E2 -13795.801} C_VEL
LIN {X 0,Y 349.55,Z 158.148,A -85,B 0,C 180,E1 -13798.851,E2 -13798.851} C_VEL
LIN {X 0,Y 347.789,Z 150.161,A -85,B 0,C 180,E1 -13800.932,E2 -13800.932} C_VEL
LIN {X 0,Y 347.745,Z 150.167,A -85,B 0,C 180,E1 -13804.463,E2 -13804.463} C_VEL
LIN {X 0,Y 347.774,Z 150.167,A -85,B 0,C 180,E1 -13807.988,E2 -13807.988} C_VEL
LIN {X 0,Y 347.751,Z 150.171,A -85,B 0,C 180,E1 -13811.829,E2 -13811.829} C_VEL
LIN {X 0,Y 347.706,Z 150.17,A -85,B 0,C 180,E1 -13815.026,E2 -13815.026} C_VEL
LIN {X 0,Y 347.75,Z 150.165,A -85,B 0,C 180,E1 -13818.396,E2 -13818.396} C_VEL
LIN {X 0,Y 347.772,Z 150.164,A -85,B 0,C 180,E1 -13822.011,E2 -13822.011} C_VEL
LIN {X 0,Y 347.743,Z 150.171,A -85,B 0,C 180,E1 -13825.535,E2 -13825.535} C_VEL
LIN {X 0,Y 347.763,Z 150.167,A -85,B 0,C 180,E1 -13829.653,E2 -13829.653} C_VEL
LIN {X 0,Y 347.851,Z 150.153,A -85,B 0,C 180,E1 -13832.744,E2 -13832.744} C_VEL
LIN {X 0,Y 347.787,Z 150.16,A -85,B 0,C 180,E1 -13836.161,E2 -13836.161} C_VEL
LIN {X 0,Y 347.804,Z 150.158,A -85,B 0,C 180,E1 -13839.908,E2 -13839.908} C_VEL
LIN {X 0,Y 347.83,Z 150.157,A -85,B 0,C 180,E1 -13843.568,E2 -13843.568} C_VEL
LIN {X 0,Y 347.888,Z 150.153,A -85,B 0,C 180,E1 -13847.16,E2 -13847.16} C_VEL
LIN {X 0,Y 347.962,Z 150.141,A -85,B 0,C 180,E1 -13850.701,E2 -13850.701} C_VEL
LIN {X 0,Y 348.09,Z 150.128,A -85,B 0,C 180,E1 -13853.041,E2 -13853.041} C_VEL
LIN {X 0,Y 348.206,Z 150.108,A -85,B 0,C 180,E1 -13857.686,E2 -13857.686} C_VEL
LIN {X 0,Y 348.365,Z 150.088,A -85,B 0,C 180,E1 -13859.999,E2 -13859.999} C_VEL
LIN {X 0,Y 348.205,Z 150.109,A -85,B 0,C 180,E1 -13862.313,E2 -13862.313} C_VEL
LIN {X 0,Y 348.089,Z 150.126,A -85,B 0,C 180,E1 -13866.957,E2 -13866.957} C_VEL
LIN {X 0,Y 347.926,Z 150.147,A -85,B 0,C 180,E1 -13870.474,E2 -13870.474} C_VEL
LIN {X 0,Y 347.895,Z 150.149,A -85,B 0,C 180,E1 -13874.149,E2 -13874.149} C_VEL
LIN {X 0,Y 347.888,Z 150.152,A -85,B 0,C 180,E1 -13878.29,E2 -13878.29} C_VEL
LIN {X 0,Y 347.785,Z 150.16,A -85,B 0,C 180,E1 -13881.635,E2 -13881.635} C_VEL
LIN {X 0,Y 347.808,Z 150.157,A -85,B 0,C 180,E1 -13885.108,E2 -13885.108} C_VEL
LIN {X 0,Y 347.806,Z 150.158,A -85,B 0,C 180,E1 -13887.693,E2 -13887.693} C_VEL
LIN {X 0,Y 347.759,Z 150.168,A -85,B 0,C 180,E1 -13890.346,E2 -13890.346} C_VEL
LIN {X 0,Y 347.739,Z 150.169,A -85,B 0,C 180,E1 -13894.464,E2 -13894.464} C_VEL
LIN {X 0,Y 347.771,Z 150.167,A -85,B 0,C 180,E1 -13897.989,E2 -13897.989} C_VEL
LIN {X 0,Y 347.782,Z 150.165,A -85,B 0,C 180,E1 -13901.825,E2 -13901.825} C_VEL
LIN {X 0,Y 347.826,Z 150.155,A -85,B 0,C 180,E1 -13905.006,E2 -13905.006} C_VEL
LIN {X 0,Y 347.781,Z 150.162,A -85,B 0,C 180,E1 -13908.39,E2 -13908.39} C_VEL
LIN {X 0,Y 347.771,Z 150.165,A -85,B 0,C 180,E1 -13912.011,E2 -13912.011} C_VEL
LIN {X 0,Y 347.739,Z 150.17,A -85,B 0,C 180,E1 -13915.536,E2 -13915.536} C_VEL
LIN {X 0,Y 347.758,Z 150.169,A -85,B 0,C 180,E1 -13919.654,E2 -13919.654} C_VEL
LIN {X 0,Y 347.846,Z 150.153,A -85,B 0,C 180,E1 -13922.745,E2 -13922.745} C_VEL
LIN {X 0,Y 347.783,Z 150.161,A -85,B 0,C 180,E1 -13926.162,E2 -13926.162} C_VEL
LIN {X 0,Y 347.812,Z 150.158,A -85,B 0,C 180,E1 -13929.91,E2 -13929.91} C_VEL
LIN {X 0,Y 347.862,Z 150.15,A -85,B 0,C 180,E1 -13932.36,E2 -13932.36} C_VEL
LIN {X 0,Y 347.893,Z 150.147,A -85,B 0,C 180,E1 -13935.971,E2 -13935.971} C_VEL
LIN {X 0,Y 347.924,Z 150.146,A -85,B 0,C 180,E1 -13939.526,E2 -13939.526} C_VEL
LIN {X 0,Y 348.07,Z 150.125,A -85,B 0,C 180,E1 -13941.875,E2 -13941.875} C_VEL
LIN {X 0,Y 348.064,Z 150.125,A -85,B 0,C 180,E1 -13944.206,E2 -13944.206} C_VEL
LIN {X 0,Y 348.205,Z 150.109,A -85,B 0,C 180,E1 -13947.687,E2 -13947.687} C_VEL
LIN {X 0,Y 348.343,Z 150.09,A -85,B 0,C 180,E1 -13950.001,E2 -13950.001} C_VEL
LIN {X 0,Y 348.205,Z 150.109,A -85,B 0,C 180,E1 -13952.314,E2 -13952.314} C_VEL
LIN {X 0,Y 348.104,Z 150.125,A -85,B 0,C 180,E1 -13956.958,E2 -13956.958} C_VEL
LIN {X 0,Y 347.965,Z 150.139,A -85,B 0,C 180,E1 -13959.299,E2 -13959.299} C_VEL
LIN {X 0,Y 347.888,Z 150.153,A -85,B 0,C 180,E1 -13962.84,E2 -13962.84} C_VEL
LIN {X 0,Y 347.962,Z 150.172,A -85,B 0,C 180,E1 -13964.128,E2 -13964.128} C_VEL
LIN {X 0,Y 348.994,Z 155.486,A -85,B 0,C 180,E1 -13965.593,E2 -13965.593} C_VEL
LIN {X 0,Y 354.618,Z 172.248,A -85,B 0,C 180,E1 -13966.308,E2 -13966.308} C_VEL
LIN {X 0,Y 356.271,Z 180.902,A -85,B 0,C 180,E1 -13966.598,E2 -13966.598} C_VEL
LIN {X 0,Y 354.467,Z 262.581,A -85,B 0,C 180,E1 -13968.357,E2 -13968.357} C_VEL
LIN {X 0,Y 353.899,Z 275.849,A -85,B 0,C 180,E1 -13968.865,E2 -13968.865} C_VEL
LIN {X 0,Y 353.267,Z 288.977,A -85,B 0,C 180,E1 -13969.617,E2 -13969.617} C_VEL
LIN {X 0,Y 352.472,Z 301.145,A -85,B 0,C 180,E1 -13970.572,E2 -13970.572} C_VEL
LIN {X 0,Y 351.441,Z 312.522,A -85,B 0,C 180,E1 -13971.714,E2 -13971.714} C_VEL
LIN {X 0,Y 350.505,Z 321.984,A -85,B 0,C 180,E1 -13972.894,E2 -13972.894} C_VEL
LIN {X 0,Y 349.587,Z 331.394,A -85,B 0,C 180,E1 -13974.339,E2 -13974.339} C_VEL
LIN {X 0,Y 348.647,Z 340.146,A -85,B 0,C 180,E1 -13976.005,E2 -13976.005} C_VEL
LIN {X 0,Y 347.919,Z 347.282,A -85,B 0,C 180,E1 -13977.685,E2 -13977.685} C_VEL
LIN {X 0,Y 347.266,Z 353.499,A -85,B 0,C 180,E1 -13979.515,E2 -13979.515} C_VEL
LIN {X 0,Y 346.9,Z 357.443,A -85,B 0,C 180,E1 -13980.985,E2 -13980.985} C_VEL
LIN {X 0,Y 346.04,Z 359.561,A -85,B 0,C 180,E1 -13981.886,E2 -13981.886} C_VEL
LIN {X 0,Y 342.864,Z 362.452,A -85,B 0,C 180,E1 -13983.374,E2 -13983.374} C_VEL
LIN {X 0,Y 340.232,Z 364.243,A -85,B 0,C 180,E1 -13984.604,E2 -13984.604} C_VEL
LIN {X 0,Y 339.078,Z 365.3,A -85,B 0,C 180,E1 -13985.572,E2 -13985.572} C_VEL
LIN {X 0,Y 338.967,Z 365.566,A -85,B 0,C 180,E1 -13985.903,E2 -13985.903} C_VEL
LIN {X 0,Y 338.932,Z 366.613,A -85,B 0,C 180,E1 -13988.006,E2 -13988.006} C_VEL
LIN {X 0,Y 339.043,Z 366.442,A -85,B 0,C 180,E1 -13989.987,E2 -13989.987} C_VEL
LIN {X 0,Y 339.243,Z 365.333,A -85,B 0,C 180,E1 -13991.773,E2 -13991.773} C_VEL
LIN {X 0,Y 339.599,Z 363.252,A -85,B 0,C 180,E1 -13993.588,E2 -13993.588} C_VEL
LIN {X 0,Y 340.041,Z 360.264,A -85,B 0,C 180,E1 -13995.356,E2 -13995.356} C_VEL
LIN {X 0,Y 340.752,Z 355.365,A -85,B 0,C 180,E1 -13997.449,E2 -13997.449} C_VEL
LIN {X 0,Y 341.705,Z 348.797,A -85,B 0,C 180,E1 -13999.553,E2 -13999.553} C_VEL
LIN {X 0,Y 342.9,Z 341.195,A -85,B 0,C 180,E1 -14001.423,E2 -14001.423} C_VEL
LIN {X 0,Y 344.076,Z 332.862,A -85,B 0,C 180,E1 -14003.072,E2 -14003.072} C_VEL
LIN {X 0,Y 345.331,Z 323.982,A -85,B 0,C 180,E1 -14004.496,E2 -14004.496} C_VEL
LIN {X 0,Y 346.581,Z 313.876,A -85,B 0,C 180,E1 -14005.806,E2 -14005.806} C_VEL
LIN {X 0,Y 347.874,Z 302.852,A -85,B 0,C 180,E1 -14006.944,E2 -14006.944} C_VEL
LIN {X 0,Y 348.926,Z 291.481,A -85,B 0,C 180,E1 -14007.87,E2 -14007.87} C_VEL
LIN {X 0,Y 349.684,Z 279.268,A -85,B 0,C 180,E1 -14008.626,E2 -14008.626} C_VEL
LIN {X 0,Y 350.353,Z 265.976,A -85,B 0,C 180,E1 -14009.182,E2 -14009.182} C_VEL
LIN {X 0,Y 351.218,Z 236.788,A -85,B 0,C 180,E1 -14009.87,E2 -14009.87} C_VEL
LIN {X 0,Y 352.655,Z 183.319,A -85,B 0,C 180,E1 -14011.061,E2 -14011.061} C_VEL
LIN {X 0,Y 351.434,Z 178.639,A -85,B 0,C 180,E1 -14011.278,E2 -14011.278} C_VEL
LIN {X 0,Y 345.685,Z 164.797,A -85,B 0,C 180,E1 -14012.122,E2 -14012.122} C_VEL
LIN {X 0,Y 342.262,Z 157.095,A -85,B 0,C 180,E1 -14012.649,E2 -14012.649} C_VEL
LIN {X 0,Y 340.803,Z 151.039,A -85,B 0,C 180,E1 -14014.575,E2 -14014.575} C_VEL
LIN {X 0,Y 340.744,Z 151.045,A -85,B 0,C 180,E1 -14018.208,E2 -14018.208} C_VEL
LIN {X 0,Y 340.796,Z 151.034,A -85,B 0,C 180,E1 -14021.982,E2 -14021.982} C_VEL
LIN {X 0,Y 340.873,Z 151.028,A -85,B 0,C 180,E1 -14025.706,E2 -14025.706} C_VEL
LIN {X 0,Y 340.852,Z 151.026,A -85,B 0,C 180,E1 -14029.306,E2 -14029.306} C_VEL
LIN {X 0,Y 341.006,Z 151.008,A -85,B 0,C 180,E1 -14032.897,E2 -14032.897} C_VEL
LIN {X 0,Y 340.818,Z 151.029,A -85,B 0,C 180,E1 -14035.269,E2 -14035.269} C_VEL
LIN {X 0,Y 341.13,Z 150.993,A -85,B 0,C 180,E1 -14037.639,E2 -14037.639} C_VEL
LIN {X 0,Y 341.093,Z 150.996,A -85,B 0,C 180,E1 -14041.181,E2 -14041.181} C_VEL
LIN {X 0,Y 341.122,Z 150.987,A -85,B 0,C 180,E1 -14042.362,E2 -14042.362} C_VEL
LIN {X 0,Y 341.019,Z 151.002,A -85,B 0,C 180,E1 -14045.915,E2 -14045.915} C_VEL
LIN {X 0,Y 340.969,Z 151.012,A -85,B 0,C 180,E1 -14048.357,E2 -14048.357} C_VEL
LIN {X 0,Y 340.838,Z 151.022,A -85,B 0,C 180,E1 -14051.9,E2 -14051.9} C_VEL
LIN {X 0,Y 340.815,Z 151.024,A -85,B 0,C 180,E1 -14054.328,E2 -14054.328} C_VEL
LIN {X 0,Y 340.754,Z 151.034,A -85,B 0,C 180,E1 -14058.422,E2 -14058.422} C_VEL
LIN {X 0,Y 340.694,Z 151.046,A -85,B 0,C 180,E1 -14061.829,E2 -14061.829} C_VEL
LIN {X 0,Y 340.709,Z 151.04,A -85,B 0,C 180,E1 -14064.821,E2 -14064.821} C_VEL
LIN {X 0,Y 340.68,Z 151.042,A -85,B 0,C 180,E1 -14068.326,E2 -14068.326} C_VEL
LIN {X 0,Y 340.695,Z 151.041,A -85,B 0,C 180,E1 -14071.046,E2 -14071.046} C_VEL
LIN {X 0,Y 340.723,Z 151.038,A -85,B 0,C 180,E1 -14075.279,E2 -14075.279} C_VEL
LIN {X 0,Y 340.699,Z 151.041,A -85,B 0,C 180,E1 -14078.382,E2 -14078.382} C_VEL
LIN {X 0,Y 340.698,Z 151.045,A -85,B 0,C 180,E1 -14082.044,E2 -14082.044} C_VEL
LIN {X 0,Y 340.656,Z 151.054,A -85,B 0,C 180,E1 -14086.227,E2 -14086.227} C_VEL
LIN {X 0,Y 340.676,Z 151.051,A -85,B 0,C 180,E1 -14088.688,E2 -14088.688} C_VEL
LIN {X 0,Y 340.724,Z 151.046,A -85,B 0,C 180,E1 -14091.771,E2 -14091.771} C_VEL
LIN {X 0,Y 340.728,Z 151.045,A -85,B 0,C 180,E1 -14095.595,E2 -14095.595} C_VEL
LIN {X 0,Y 340.71,Z 151.158,A -85,B 0,C 180,E1 -14097.171,E2 -14097.171} C_VEL
LIN {X 0,Y 343.436,Z 162.042,A -85,B 0,C 180,E1 -14100.301,E2 -14100.301} C_VEL
LIN {X 0,Y 345.548,Z 172.405,A -85,B 0,C 180,E1 -14103.093,E2 -14103.093} C_VEL
LIN {X 0,Y 345.803,Z 174.593,A -85,B 0,C 180,E1 -14103.649,E2 -14103.649} C_VEL
LIN {X 0,Y 344.866,Z 183.05,A -85,B 0,C 180,E1 -14105.622,E2 -14105.622} C_VEL
LIN {X 0,Y 349.049,Z 205.13,A -85,B 0,C 180,E1 -14106.547,E2 -14106.547} C_VEL
LIN {X 0,Y 351.653,Z 223.565,A -85,B 0,C 180,E1 -14107.213,E2 -14107.213} C_VEL
LIN {X 0,Y 349.964,Z 292.711,A -85,B 0,C 180,E1 -14108.776,E2 -14108.776} C_VEL
LIN {X 0,Y 349.086,Z 306.88,A -85,B 0,C 180,E1 -14109.331,E2 -14109.331} C_VEL
LIN {X 0,Y 348.052,Z 318.552,A -85,B 0,C 180,E1 -14110,E2 -14110} C_VEL
LIN {X 0,Y 346.746,Z 330.522,A -85,B 0,C 180,E1 -14110.923,E2 -14110.923} C_VEL
LIN {X 0,Y 345.332,Z 342.021,A -85,B 0,C 180,E1 -14112.072,E2 -14112.072} C_VEL
LIN {X 0,Y 343.944,Z 352.435,A -85,B 0,C 180,E1 -14113.376,E2 -14113.376} C_VEL
LIN {X 0,Y 342.735,Z 361.829,A -85,B 0,C 180,E1 -14114.843,E2 -14114.843} C_VEL
LIN {X 0,Y 341.502,Z 370.96,A -85,B 0,C 180,E1 -14116.613,E2 -14116.613} C_VEL
LIN {X 0,Y 340.437,Z 378.345,A -85,B 0,C 180,E1 -14118.387,E2 -14118.387} C_VEL
LIN {X 0,Y 339.895,Z 383.364,A -85,B 0,C 180,E1 -14119.877,E2 -14119.877} C_VEL
LIN {X 0,Y 339.438,Z 388.264,A -85,B 0,C 180,E1 -14121.666,E2 -14121.666} C_VEL
LIN {X 0,Y 339.155,Z 392.036,A -85,B 0,C 180,E1 -14123.455,E2 -14123.455} C_VEL
LIN {X 0,Y 339.07,Z 394.782,A -85,B 0,C 180,E1 -14125.244,E2 -14125.244} C_VEL
LIN {X 0,Y 339.089,Z 396.092,A -85,B 0,C 180,E1 -14126.434,E2 -14126.434} C_VEL
LIN {X 0,Y 339.069,Z 396.976,A -85,B 0,C 180,E1 -14127.623,E2 -14127.623} C_VEL
LIN {X 0,Y 339.161,Z 397.427,A -85,B 0,C 180,E1 -14128.812,E2 -14128.812} C_VEL
LIN {X 0,Y 339.229,Z 397.481,A -85,B 0,C 180,E1 -14129.999,E2 -14129.999} C_VEL
LIN {X 0,Y 339.167,Z 397.133,A -85,B 0,C 180,E1 -14131.187,E2 -14131.187} C_VEL
LIN {X 0,Y 339.086,Z 396.363,A -85,B 0,C 180,E1 -14132.375,E2 -14132.375} C_VEL
LIN {X 0,Y 339.097,Z 395.147,A -85,B 0,C 180,E1 -14133.564,E2 -14133.564} C_VEL
LIN {X 0,Y 339.095,Z 393.514,A -85,B 0,C 180,E1 -14134.755,E2 -14134.755} C_VEL
LIN {X 0,Y 339.173,Z 390.205,A -85,B 0,C 180,E1 -14136.543,E2 -14136.543} C_VEL
LIN {X 0,Y 339.416,Z 385.794,A -85,B 0,C 180,E1 -14138.333,E2 -14138.333} C_VEL
LIN {X 0,Y 339.822,Z 380.155,A -85,B 0,C 180,E1 -14140.124,E2 -14140.124} C_VEL
LIN {X 0,Y 340.477,Z 373.095,A -85,B 0,C 180,E1 -14141.912,E2 -14141.912} C_VEL
LIN {X 0,Y 341.383,Z 364.226,A -85,B 0,C 180,E1 -14143.694,E2 -14143.694} C_VEL
LIN {X 0,Y 342.387,Z 354.573,A -85,B 0,C 180,E1 -14145.257,E2 -14145.257} C_VEL
LIN {X 0,Y 343.515,Z 343.855,A -85,B 0,C 180,E1 -14146.643,E2 -14146.643} C_VEL
LIN {X 0,Y 344.688,Z 332.46,A -85,B 0,C 180,E1 -14147.808,E2 -14147.808} C_VEL
LIN {X 0,Y 345.699,Z 320.654,A -85,B 0,C 180,E1 -14148.751,E2 -14148.751} C_VEL
LIN {X 0,Y 346.693,Z 307.765,A -85,B 0,C 180,E1 -14149.502,E2 -14149.502} C_VEL
LIN {X 0,Y 347.355,Z 294.16,A -85,B 0,C 180,E1 -14150.04,E2 -14150.04} C_VEL
LIN {X 0,Y 348.827,Z 222.739,A -85,B 0,C 180,E1 -14151.629,E2 -14151.629} C_VEL
LIN {X 0,Y 343.453,Z 185.024,A -85,B 0,C 180,E1 -14152.825,E2 -14152.825} C_VEL
LIN {X 0,Y 344.828,Z 172.249,A -85,B 0,C 180,E1 -14155.776,E2 -14155.776} C_VEL
LIN {X 0,Y 343.834,Z 165.836,A -85,B 0,C 180,E1 -14157.38,E2 -14157.38} C_VEL
LIN {X 0,Y 341.61,Z 154.868,A -85,B 0,C 180,E1 -14160.222,E2 -14160.222} C_VEL
LIN {X 0,Y 340.718,Z 151.041,A -85,B 0,C 180,E1 -14161.301,E2 -14161.301} C_VEL
LIN {X 0,Y 340.719,Z 151.041,A -85,B 0,C 180,E1 -14165.278,E2 -14165.278} C_VEL
LIN {X 0,Y 340.71,Z 151.043,A -85,B 0,C 180,E1 -14168.385,E2 -14168.385} C_VEL
LIN {X 0,Y 340.699,Z 151.047,A -85,B 0,C 180,E1 -14172.045,E2 -14172.045} C_VEL
LIN {X 0,Y 340.652,Z 151.05,A -85,B 0,C 180,E1 -14176.226,E2 -14176.226} C_VEL
LIN {X 0,Y 340.688,Z 151.049,A -85,B 0,C 180,E1 -14179.752,E2 -14179.752} C_VEL
LIN {X 0,Y 340.704,Z 151.045,A -85,B 0,C 180,E1 -14183.258,E2 -14183.258} C_VEL
LIN {X 0,Y 340.691,Z 151.045,A -85,B 0,C 180,E1 -14186.153,E2 -14186.153} C_VEL
LIN {X 0,Y 340.774,Z 151.034,A -85,B 0,C 180,E1 -14190.332,E2 -14190.332} C_VEL
LIN {X 0,Y 340.804,Z 151.032,A -85,B 0,C 180,E1 -14193.019,E2 -14193.019} C_VEL
LIN {X 0,Y 340.727,Z 151.042,A -85,B 0,C 180,E1 -14196.926,E2 -14196.926} C_VEL
LIN {X 0,Y 340.758,Z 151.037,A -85,B 0,C 180,E1 -14200.731,E2 -14200.731} C_VEL
LIN {X 0,Y 340.815,Z 151.029,A -85,B 0,C 180,E1 -14204.45,E2 -14204.45} C_VEL
LIN {X 0,Y 340.848,Z 151.024,A -85,B 0,C 180,E1 -14208.1,E2 -14208.1} C_VEL
LIN {X 0,Y 341.036,Z 151.001,A -85,B 0,C 180,E1 -14211.705,E2 -14211.705} C_VEL
LIN {X 0,Y 341.036,Z 151.001,A -85,B 0,C 180,E1 -14214.085,E2 -14214.085} C_VEL
LIN {X 0,Y 341.168,Z 150.985,A -85,B 0,C 180,E1 -14217.638,E2 -14217.638} C_VEL
LIN {X 0,Y 341.314,Z 150.966,A -85,B 0,C 180,E1 -14219.999,E2 -14219.999} C_VEL
LIN {X 0,Y 341.167,Z 150.986,A -85,B 0,C 180,E1 -14222.361,E2 -14222.361} C_VEL
LIN {X 0,Y 341.057,Z 151,A -85,B 0,C 180,E1 -14227.101,E2 -14227.101} C_VEL
LIN {X 0,Y 340.868,Z 151.027,A -85,B 0,C 180,E1 -14230.693,E2 -14230.693} C_VEL
LIN {X 0,Y 340.859,Z 151.027,A -85,B 0,C 180,E1 -14234.324,E2 -14234.324} C_VEL
LIN {X 0,Y 340.834,Z 151.032,A -85,B 0,C 180,E1 -14238.466,E2 -14238.466} C_VEL
LIN {X 0,Y 340.749,Z 151.038,A -85,B 0,C 180,E1 -14241.856,E2 -14241.856} C_VEL
LIN {X 0,Y 340.768,Z 151.035,A -85,B 0,C 180,E1 -14245.664,E2 -14245.664} C_VEL
LIN {X 0,Y 340.737,Z 151.044,A -85,B 0,C 180,E1 -14248.319,E2 -14248.319} C_VEL
LIN {X 0,Y 340.699,Z 151.043,A -85,B 0,C 180,E1 -14251.044,E2 -14251.044} C_VEL
LIN {X 0,Y 340.714,Z 151.041,A -85,B 0,C 180,E1 -14255.279,E2 -14255.279} C_VEL
LIN {X 0,Y 340.713,Z 151.044,A -85,B 0,C 180,E1 -14258.388,E2 -14258.388} C_VEL
LIN {X 0,Y 340.722,Z 151.04,A -85,B 0,C 180,E1 -14261.303,E2 -14261.303} C_VEL
LIN {X 0,Y 340.777,Z 151.034,A -85,B 0,C 180,E1 -14264.522,E2 -14264.522} C_VEL
LIN {X 0,Y 340.749,Z 151.042,A -85,B 0,C 180,E1 -14267.944,E2 -14267.944} C_VEL
LIN {X 0,Y 340.729,Z 151.041,A -85,B 0,C 180,E1 -14270.253,E2 -14270.253} C_VEL
LIN {X 0,Y 340.706,Z 151.046,A -85,B 0,C 180,E1 -14273.559,E2 -14273.559} C_VEL
LIN {X 0,Y 340.688,Z 151.046,A -85,B 0,C 180,E1 -14276.154,E2 -14276.154} C_VEL
LIN {X 0,Y 340.769,Z 151.034,A -85,B 0,C 180,E1 -14280.333,E2 -14280.333} C_VEL
LIN {X 0,Y 340.8,Z 151.032,A -85,B 0,C 180,E1 -14283.02,E2 -14283.02} C_VEL
LIN {X 0,Y 340.724,Z 151.041,A -85,B 0,C 180,E1 -14286.928,E2 -14286.928} C_VEL
LIN {X 0,Y 340.79,Z 151.032,A -85,B 0,C 180,E1 -14290.734,E2 -14290.734} C_VEL
LIN {X 0,Y 340.782,Z 151.037,A -85,B 0,C 180,E1 -14293.219,E2 -14293.219} C_VEL
LIN {X 0,Y 340.84,Z 151.028,A -85,B 0,C 180,E1 -14296.891,E2 -14296.891} C_VEL
LIN {X 0,Y 340.924,Z 151.015,A -85,B 0,C 180,E1 -14300.508,E2 -14300.508} C_VEL
LIN {X 0,Y 341.072,Z 151,A -85,B 0,C 180,E1 -14302.899,E2 -14302.899} C_VEL
LIN {X 0,Y 341.166,Z 150.986,A -85,B 0,C 180,E1 -14307.639,E2 -14307.639} C_VEL
LIN {X 0,Y 341.293,Z 150.969,A -85,B 0,C 180,E1 -14310.001,E2 -14310.001} C_VEL
LIN {X 0,Y 341.167,Z 150.986,A -85,B 0,C 180,E1 -14312.362,E2 -14312.362} C_VEL
LIN {X 0,Y 341.073,Z 151,A -85,B 0,C 180,E1 -14317.103,E2 -14317.103} C_VEL
LIN {X 0,Y 340.868,Z 151.027,A -85,B 0,C 180,E1 -14320.695,E2 -14320.695} C_VEL
LIN {X 0,Y 340.911,Z 151.182,A -85,B 0,C 180,E1 -14323.869,E2 -14323.869} C_VEL
LIN {X 0,Y 341.81,Z 155.556,A -85,B 0,C 180,E1 -14325.144,E2 -14325.144} C_VEL
LIN {X 0,Y 348.119,Z 174.284,A -85,B 0,C 180,E1 -14325.978,E2 -14325.978} C_VEL
LIN {X 0,Y 349.511,Z 181.119,A -85,B 0,C 180,E1 -14326.218,E2 -14326.218} C_VEL
LIN {X 0,Y 347.674,Z 263.469,A -85,B 0,C 180,E1 -14328.039,E2 -14328.039} C_VEL
LIN {X 0,Y 347.093,Z 277.594,A -85,B 0,C 180,E1 -14328.61,E2 -14328.61} C_VEL
LIN {X 0,Y 346.426,Z 289.613,A -85,B 0,C 180,E1 -14329.326,E2 -14329.326} C_VEL
LIN {X 0,Y 345.572,Z 302.248,A -85,B 0,C 180,E1 -14330.351,E2 -14330.351} C_VEL
LIN {X 0,Y 344.463,Z 313.78,A -85,B 0,C 180,E1 -14331.547,E2 -14331.547} C_VEL
LIN {X 0,Y 343.415,Z 324.325,A -85,B 0,C 180,E1 -14332.94,E2 -14332.94} C_VEL
LIN {X 0,Y 342.341,Z 334.173,A -85,B 0,C 180,E1 -14334.558,E2 -14334.558} C_VEL
LIN {X 0,Y 341.464,Z 342.506,A -85,B 0,C 180,E1 -14336.265,E2 -14336.265} C_VEL
LIN {X 0,Y 340.753,Z 348.947,A -85,B 0,C 180,E1 -14337.896,E2 -14337.896} C_VEL
LIN {X 0,Y 340.119,Z 354.914,A -85,B 0,C 180,E1 -14339.791,E2 -14339.791} C_VEL
LIN {X 0,Y 339.594,Z 360.095,A -85,B 0,C 180,E1 -14341.952,E2 -14341.952} C_VEL
LIN {X 0,Y 339.217,Z 363.577,A -85,B 0,C 180,E1 -14344.033,E2 -14344.033} C_VEL
LIN {X 0,Y 338.967,Z 365.566,A -85,B 0,C 180,E1 -14345.903,E2 -14345.903} C_VEL
LIN {X 0,Y 338.258,Z 366.291,A -85,B 0,C 180,E1 -14346.889,E2 -14346.889} C_VEL
LIN {X 0,Y 335.421,Z 366.959,A -85,B 0,C 180,E1 -14348.503,E2 -14348.503} C_VEL
LIN {X 0,Y 333.084,Z 366.903,A -85,B 0,C 180,E1 -14349.811,E2 -14349.811} C_VEL
LIN {X 0,Y 332.13,Z 366.45,A -85,B 0,C 180,E1 -14350.819,E2 -14350.819} C_VEL
LIN {X 0,Y 332.077,Z 366.211,A -85,B 0,C 180,E1 -14351.158,E2 -14351.158} C_VEL
LIN {X 0,Y 332.291,Z 365.036,A -85,B 0,C 180,E1 -14352.595,E2 -14352.595} C_VEL
LIN {X 0,Y 332.882,Z 361.627,A -85,B 0,C 180,E1 -14355.014,E2 -14355.014} C_VEL
LIN {X 0,Y 333.531,Z 357.342,A -85,B 0,C 180,E1 -14357.075,E2 -14357.075} C_VEL
LIN {X 0,Y 334.45,Z 351.471,A -85,B 0,C 180,E1 -14359.157,E2 -14359.157} C_VEL
LIN {X 0,Y 335.597,Z 344.458,A -85,B 0,C 180,E1 -14361.08,E2 -14361.08} C_VEL
LIN {X 0,Y 336.742,Z 336.851,A -85,B 0,C 180,E1 -14362.754,E2 -14362.754} C_VEL
LIN {X 0,Y 338.003,Z 328.856,A -85,B 0,C 180,E1 -14364.187,E2 -14364.187} C_VEL
LIN {X 0,Y 339.295,Z 319.223,A -85,B 0,C 180,E1 -14365.603,E2 -14365.603} C_VEL
LIN {X 0,Y 340.694,Z 308.47,A -85,B 0,C 180,E1 -14366.864,E2 -14366.864} C_VEL
LIN {X 0,Y 341.934,Z 296.717,A -85,B 0,C 180,E1 -14367.959,E2 -14367.959} C_VEL
LIN {X 0,Y 342.976,Z 284.111,A -85,B 0,C 180,E1 -14368.843,E2 -14368.843} C_VEL
LIN {X 0,Y 343.695,Z 271.674,A -85,B 0,C 180,E1 -14369.469,E2 -14369.469} C_VEL
LIN {X 0,Y 344.275,Z 258.511,A -85,B 0,C 180,E1 -14369.886,E2 -14369.886} C_VEL
LIN {X 0,Y 346.343,Z 184.518,A -85,B 0,C 180,E1 -14371.563,E2 -14371.563} C_VEL
LIN {X 0,Y 344.522,Z 178.853,A -85,B 0,C 180,E1 -14371.865,E2 -14371.865} C_VEL
LIN {X 0,Y 337.633,Z 162.988,A -85,B 0,C 180,E1 -14372.914,E2 -14372.914} C_VEL
LIN {X 0,Y 335.11,Z 157.496,A -85,B 0,C 180,E1 -14373.325,E2 -14373.325} C_VEL
LIN {X 0,Y 333.753,Z 151.918,A -85,B 0,C 180,E1 -14375.177,E2 -14375.177} C_VEL
LIN {X 0,Y 333.673,Z 151.923,A -85,B 0,C 180,E1 -14379.02,E2 -14379.02} C_VEL
LIN {X 0,Y 333.744,Z 151.913,A -85,B 0,C 180,E1 -14381.587,E2 -14381.587} C_VEL
LIN {X 0,Y 333.812,Z 151.908,A -85,B 0,C 180,E1 -14385.578,E2 -14385.578} C_VEL
LIN {X 0,Y 333.822,Z 151.903,A -85,B 0,C 180,E1 -14389.078,E2 -14389.078} C_VEL
LIN {X 0,Y 333.961,Z 151.885,A -85,B 0,C 180,E1 -14392.747,E2 -14392.747} C_VEL
LIN {X 0,Y 333.784,Z 151.905,A -85,B 0,C 180,E1 -14395.169,E2 -14395.169} C_VEL
LIN {X 0,Y 334.071,Z 151.873,A -85,B 0,C 180,E1 -14397.589,E2 -14397.589} C_VEL
LIN {X 0,Y 334.064,Z 151.872,A -85,B 0,C 180,E1 -14401.206,E2 -14401.206} C_VEL
LIN {X 0,Y 334.063,Z 151.865,A -85,B 0,C 180,E1 -14402.412,E2 -14402.412} C_VEL
LIN {X 0,Y 333.993,Z 151.875,A -85,B 0,C 180,E1 -14406.04,E2 -14406.04} C_VEL
LIN {X 0,Y 333.918,Z 151.89,A -85,B 0,C 180,E1 -14408.473,E2 -14408.473} C_VEL
LIN {X 0,Y 333.777,Z 151.904,A -85,B 0,C 180,E1 -14412.156,E2 -14412.156} C_VEL
LIN {X 0,Y 333.737,Z 151.905,A -85,B 0,C 180,E1 -14414.638,E2 -14414.638} C_VEL
LIN {X 0,Y 333.693,Z 151.913,A -85,B 0,C 180,E1 -14418.6,E2 -14418.6} C_VEL
LIN {X 0,Y 333.625,Z 151.925,A -85,B 0,C 180,E1 -14422.284,E2 -14422.284} C_VEL
LIN {X 0,Y 333.66,Z 151.92,A -85,B 0,C 180,E1 -14425.077,E2 -14425.077} C_VEL
LIN {X 0,Y 333.633,Z 151.923,A -85,B 0,C 180,E1 -14428.98,E2 -14428.98} C_VEL
LIN {X 0,Y 333.648,Z 151.921,A -85,B 0,C 180,E1 -14432.587,E2 -14432.587} C_VEL
LIN {X 0,Y 333.68,Z 151.918,A -85,B 0,C 180,E1 -14436.139,E2 -14436.139} C_VEL
LIN {X 0,Y 333.625,Z 151.927,A -85,B 0,C 180,E1 -14439.196,E2 -14439.196} C_VEL
LIN {X 0,Y 333.633,Z 151.928,A -85,B 0,C 180,E1 -14442.499,E2 -14442.499} C_VEL
LIN {X 0,Y 333.6,Z 151.934,A -85,B 0,C 180,E1 -14445.955,E2 -14445.955} C_VEL
LIN {X 0,Y 333.607,Z 151.933,A -85,B 0,C 180,E1 -14449.324,E2 -14449.324} C_VEL
LIN {X 0,Y 333.668,Z 151.923,A -85,B 0,C 180,E1 -14453.168,E2 -14453.168} C_VEL
LIN {X 0,Y 333.685,Z 151.973,A -85,B 0,C 180,E1 -14456.571,E2 -14456.571} C_VEL
LIN {X 0,Y 336.481,Z 163.23,A -85,B 0,C 180,E1 -14459.914,E2 -14459.914} C_VEL
LIN {X 0,Y 338.655,Z 173.799,A -85,B 0,C 180,E1 -14462.834,E2 -14462.834} C_VEL
LIN {X 0,Y 338.884,Z 176.868,A -85,B 0,C 180,E1 -14463.626,E2 -14463.626} C_VEL
LIN {X 0,Y 338.243,Z 182.94,A -85,B 0,C 180,E1 -14465.037,E2 -14465.037} C_VEL
LIN {X 0,Y 342.784,Z 206.675,A -85,B 0,C 180,E1 -14466.057,E2 -14466.057} C_VEL
LIN {X 0,Y 345.29,Z 225.041,A -85,B 0,C 180,E1 -14466.732,E2 -14466.732} C_VEL
LIN {X 0,Y 343.493,Z 292.398,A -85,B 0,C 180,E1 -14468.288,E2 -14468.288} C_VEL
LIN {X 0,Y 342.637,Z 306.301,A -85,B 0,C 180,E1 -14468.845,E2 -14468.845} C_VEL
LIN {X 0,Y 341.553,Z 317.997,A -85,B 0,C 180,E1 -14469.524,E2 -14469.524} C_VEL
LIN {X 0,Y 340.28,Z 329.226,A -85,B 0,C 180,E1 -14470.389,E2 -14470.389} C_VEL
LIN {X 0,Y 338.761,Z 340.903,A -85,B 0,C 180,E1 -14471.555,E2 -14471.555} C_VEL
LIN {X 0,Y 337.281,Z 351.451,A -85,B 0,C 180,E1 -14472.882,E2 -14472.882} C_VEL
LIN {X 0,Y 336.125,Z 360.104,A -85,B 0,C 180,E1 -14474.227,E2 -14474.227} C_VEL
LIN {X 0,Y 334.989,Z 368.112,A -85,B 0,C 180,E1 -14475.728,E2 -14475.728} C_VEL
LIN {X 0,Y 333.801,Z 375.964,A -85,B 0,C 180,E1 -14477.536,E2 -14477.536} C_VEL
LIN {X 0,Y 332.868,Z 383.215,A -85,B 0,C 180,E1 -14479.661,E2 -14479.661} C_VEL
LIN {X 0,Y 332.371,Z 388.069,A -85,B 0,C 180,E1 -14481.487,E2 -14481.487} C_VEL
LIN {X 0,Y 332.072,Z 391.803,A -85,B 0,C 180,E1 -14483.315,E2 -14483.315} C_VEL
LIN {X 0,Y 331.977,Z 394.517,A -85,B 0,C 180,E1 -14485.142,E2 -14485.142} C_VEL
LIN {X 0,Y 332.012,Z 395.815,A -85,B 0,C 180,E1 -14486.358,E2 -14486.358} C_VEL
LIN {X 0,Y 331.982,Z 396.67,A -85,B 0,C 180,E1 -14487.573,E2 -14487.573} C_VEL
LIN {X 0,Y 332.063,Z 397.107,A -85,B 0,C 180,E1 -14488.787,E2 -14488.787} C_VEL
LIN {X 0,Y 332.136,Z 397.147,A -85,B 0,C 180,E1 -14489.999,E2 -14489.999} C_VEL
LIN {X 0,Y 332.07,Z 396.785,A -85,B 0,C 180,E1 -14491.212,E2 -14491.212} C_VEL
LIN {X 0,Y 331.997,Z 395.983,A -85,B 0,C 180,E1 -14492.426,E2 -14492.426} C_VEL
LIN {X 0,Y 332.021,Z 394.752,A -85,B 0,C 180,E1 -14493.64,E2 -14493.64} C_VEL
LIN {X 0,Y 332.034,Z 391.463,A -85,B 0,C 180,E1 -14495.825,E2 -14495.825} C_VEL
LIN {X 0,Y 332.249,Z 386.942,A -85,B 0,C 180,E1 -14497.902,E2 -14497.902} C_VEL
LIN {X 0,Y 332.714,Z 380.651,A -85,B 0,C 180,E1 -14500.035,E2 -14500.035} C_VEL
LIN {X 0,Y 333.32,Z 373.778,A -85,B 0,C 180,E1 -14501.863,E2 -14501.863} C_VEL
LIN {X 0,Y 334.115,Z 366.767,A -85,B 0,C 180,E1 -14503.378,E2 -14503.378} C_VEL
LIN {X 0,Y 335.07,Z 358.454,A -85,B 0,C 180,E1 -14504.864,E2 -14504.864} C_VEL
LIN {X 0,Y 336.001,Z 349.056,A -85,B 0,C 180,E1 -14506.245,E2 -14506.245} C_VEL
LIN {X 0,Y 337.243,Z 337.562,A -85,B 0,C 180,E1 -14507.588,E2 -14507.588} C_VEL
LIN {X 0,Y 338.35,Z 326.308,A -85,B 0,C 180,E1 -14508.624,E2 -14508.624} C_VEL
LIN {X 0,Y 339.406,Z 313.706,A -85,B 0,C 180,E1 -14509.505,E2 -14509.505} C_VEL
LIN {X 0,Y 340.263,Z 300.359,A -85,B 0,C 180,E1 -14510.161,E2 -14510.161} C_VEL
LIN {X 0,Y 340.808,Z 287.701,A -85,B 0,C 180,E1 -14510.555,E2 -14510.555} C_VEL
LIN {X 0,Y 342.103,Z 223.642,A -85,B 0,C 180,E1 -14511.985,E2 -14511.985} C_VEL
LIN {X 0,Y 336.621,Z 184.622,A -85,B 0,C 180,E1 -14513.271,E2 -14513.271} C_VEL
LIN {X 0,Y 337.872,Z 173.468,A -85,B 0,C 180,E1 -14515.9,E2 -14515.9} C_VEL
LIN {X 0,Y 336.781,Z 166.549,A -85,B 0,C 180,E1 -14517.665,E2 -14517.665} C_VEL
LIN {X 0,Y 334.554,Z 155.745,A -85,B 0,C 180,E1 -14520.537,E2 -14520.537} C_VEL
LIN {X 0,Y 333.701,Z 151.917,A -85,B 0,C 180,E1 -14521.601,E2 -14521.601} C_VEL
LIN {X 0,Y 333.686,Z 151.917,A -85,B 0,C 180,E1 -14524.773,E2 -14524.773} C_VEL
LIN {X 0,Y 333.653,Z 151.924,A -85,B 0,C 180,E1 -14527.65,E2 -14527.65} C_VEL
LIN {X 0,Y 333.647,Z 151.921,A -85,B 0,C 180,E1 -14530.767,E2 -14530.767} C_VEL
LIN {X 0,Y 333.593,Z 151.93,A -85,B 0,C 180,E1 -14534.25,E2 -14534.25} C_VEL
LIN {X 0,Y 333.641,Z 151.927,A -85,B 0,C 180,E1 -14537.618,E2 -14537.618} C_VEL
LIN {X 0,Y 333.652,Z 151.923,A -85,B 0,C 180,E1 -14541.201,E2 -14541.201} C_VEL
LIN {X 0,Y 333.675,Z 151.921,A -85,B 0,C 180,E1 -14543.86,E2 -14543.86} C_VEL
LIN {X 0,Y 333.642,Z 151.927,A -85,B 0,C 180,E1 -14547.412,E2 -14547.412} C_VEL
LIN {X 0,Y 333.71,Z 151.915,A -85,B 0,C 180,E1 -14551.027,E2 -14551.027} C_VEL
LIN {X 0,Y 333.735,Z 151.913,A -85,B 0,C 180,E1 -14553.753,E2 -14553.753} C_VEL
LIN {X 0,Y 333.718,Z 151.913,A -85,B 0,C 180,E1 -14557.913,E2 -14557.913} C_VEL
LIN {X 0,Y 333.739,Z 151.912,A -85,B 0,C 180,E1 -14561.586,E2 -14561.586} C_VEL
LIN {X 0,Y 333.806,Z 151.903,A -85,B 0,C 180,E1 -14565.576,E2 -14565.576} C_VEL
LIN {X 0,Y 333.832,Z 151.904,A -85,B 0,C 180,E1 -14569.077,E2 -14569.077} C_VEL
LIN {X 0,Y 334.01,Z 151.879,A -85,B 0,C 180,E1 -14572.747,E2 -14572.747} C_VEL
LIN {X 0,Y 333.808,Z 151.905,A -85,B 0,C 180,E1 -14575.168,E2 -14575.168} C_VEL
LIN {X 0,Y 334.105,Z 151.865,A -85,B 0,C 180,E1 -14577.588,E2 -14577.588} C_VEL
LIN {X 0,Y 334.264,Z 151.844,A -85,B 0,C 180,E1 -14579.999,E2 -14579.999} C_VEL
LIN {X 0,Y 334.104,Z 151.866,A -85,B 0,C 180,E1 -14582.411,E2 -14582.411} C_VEL
LIN {X 0,Y 333.992,Z 151.877,A -85,B 0,C 180,E1 -14586.599,E2 -14586.599} C_VEL
LIN {X 0,Y 333.858,Z 151.895,A -85,B 0,C 180,E1 -14589.695,E2 -14589.695} C_VEL
LIN {X 0,Y 333.793,Z 151.903,A -85,B 0,C 180,E1 -14593.391,E2 -14593.391} C_VEL
LIN {X 0,Y 333.743,Z 151.91,A -85,B 0,C 180,E1 -14597.146,E2 -14597.146} C_VEL
LIN {X 0,Y 333.738,Z 151.91,A -85,B 0,C 180,E1 -14599.689,E2 -14599.689} C_VEL
LIN {X 0,Y 333.677,Z 151.918,A -85,B 0,C 180,E1 -14603.589,E2 -14603.589} C_VEL
LIN {X 0,Y 333.731,Z 151.916,A -85,B 0,C 180,E1 -14606.246,E2 -14606.246} C_VEL
LIN {X 0,Y 333.706,Z 151.914,A -85,B 0,C 180,E1 -14608.972,E2 -14608.972} C_VEL
LIN {X 0,Y 333.641,Z 151.924,A -85,B 0,C 180,E1 -14612.587,E2 -14612.587} C_VEL
LIN {X 0,Y 333.672,Z 151.924,A -85,B 0,C 180,E1 -14616.139,E2 -14616.139} C_VEL
LIN {X 0,Y 333.679,Z 151.917,A -85,B 0,C 180,E1 -14619.187,E2 -14619.187} C_VEL
LIN {X 0,Y 333.7,Z 151.916,A -85,B 0,C 180,E1 -14622.513,E2 -14622.513} C_VEL
LIN {X 0,Y 333.725,Z 151.917,A -85,B 0,C 180,E1 -14625.977,E2 -14625.977} C_VEL
LIN {X 0,Y 333.697,Z 151.916,A -85,B 0,C 180,E1 -14629.304,E2 -14629.304} C_VEL
LIN {X 0,Y 333.661,Z 151.921,A -85,B 0,C 180,E1 -14633.168,E2 -14633.168} C_VEL
LIN {X 0,Y 333.633,Z 151.923,A -85,B 0,C 180,E1 -14636.792,E2 -14636.792} C_VEL
LIN {X 0,Y 333.697,Z 151.92,A -85,B 0,C 180,E1 -14639.71,E2 -14639.71} C_VEL
LIN {X 0,Y 333.738,Z 151.91,A -85,B 0,C 180,E1 -14642.401,E2 -14642.401} C_VEL
LIN {X 0,Y 333.722,Z 151.914,A -85,B 0,C 180,E1 -14645.091,E2 -14645.091} C_VEL
LIN {X 0,Y 333.677,Z 151.92,A -85,B 0,C 180,E1 -14649.02,E2 -14649.02} C_VEL
LIN {X 0,Y 333.79,Z 151.907,A -85,B 0,C 180,E1 -14651.59,E2 -14651.59} C_VEL
LIN {X 0,Y 333.804,Z 151.905,A -85,B 0,C 180,E1 -14655.577,E2 -14655.577} C_VEL
LIN {X 0,Y 333.829,Z 151.903,A -85,B 0,C 180,E1 -14659.079,E2 -14659.079} C_VEL
LIN {X 0,Y 334.022,Z 151.877,A -85,B 0,C 180,E1 -14662.748,E2 -14662.748} C_VEL
LIN {X 0,Y 333.809,Z 151.906,A -85,B 0,C 180,E1 -14665.17,E2 -14665.17} C_VEL
LIN {X 0,Y 334.104,Z 151.866,A -85,B 0,C 180,E1 -14667.59,E2 -14667.59} C_VEL
LIN {X 0,Y 334.244,Z 151.847,A -85,B 0,C 180,E1 -14670.001,E2 -14670.001} C_VEL
LIN {X 0,Y 334.104,Z 151.866,A -85,B 0,C 180,E1 -14672.412,E2 -14672.412} C_VEL
LIN {X 0,Y 334.023,Z 151.877,A -85,B 0,C 180,E1 -14677.253,E2 -14677.253} C_VEL
LIN {X 0,Y 333.831,Z 151.904,A -85,B 0,C 180,E1 -14680.923,E2 -14680.923} C_VEL
LIN {X 0,Y 333.838,Z 151.915,A -85,B 0,C 180,E1 -14683.52,E2 -14683.52} C_VEL
LIN {X 0,Y 334.658,Z 155.923,A -85,B 0,C 180,E1 -14684.714,E2 -14684.714} C_VEL
LIN {X 0,Y 341.753,Z 176.838,A -85,B 0,C 180,E1 -14685.657,E2 -14685.657} C_VEL
LIN {X 0,Y 342.859,Z 182.51,A -85,B 0,C 180,E1 -14685.858,E2 -14685.858} C_VEL
LIN {X 0,Y 340.922,Z 264.157,A -85,B 0,C 180,E1 -14687.703,E2 -14687.703} C_VEL
LIN {X 0,Y 340.302,Z 277.903,A -85,B 0,C 180,E1 -14688.27,E2 -14688.27} C_VEL
LIN {X 0,Y 339.597,Z 290.413,A -85,B 0,C 180,E1 -14689.038,E2 -14689.038} C_VEL
LIN {X 0,Y 338.747,Z 302.284,A -85,B 0,C 180,E1 -14690.019,E2 -14690.019} C_VEL
LIN {X 0,Y 337.657,Z 313.404,A -85,B 0,C 180,E1 -14691.185,E2 -14691.185} C_VEL
LIN {X 0,Y 336.562,Z 323.719,A -85,B 0,C 180,E1 -14692.543,E2 -14692.543} C_VEL
LIN {X 0,Y 335.523,Z 333.25,A -85,B 0,C 180,E1 -14694.109,E2 -14694.109} C_VEL
LIN {X 0,Y 334.597,Z 341.527,A -85,B 0,C 180,E1 -14695.782,E2 -14695.782} C_VEL
LIN {X 0,Y 333.771,Z 348.775,A -85,B 0,C 180,E1 -14697.597,E2 -14697.597} C_VEL
LIN {X 0,Y 333.102,Z 354.874,A -85,B 0,C 180,E1 -14699.541,E2 -14699.541} C_VEL
LIN {X 0,Y 332.673,Z 358.935,A -85,B 0,C 180,E1 -14701.171,E2 -14701.171} C_VEL
LIN {X 0,Y 332.264,Z 362.977,A -85,B 0,C 180,E1 -14703.364,E2 -14703.364} C_VEL
LIN {X 0,Y 332.004,Z 364.937,A -85,B 0,C 180,E1 -14704.859,E2 -14704.859} C_VEL
LIN {X 0,Y 331.838,Z 366.254,A -85,B 0,C 180,E1 -14706.41,E2 -14706.41} C_VEL
LIN {X 0,Y 331.865,Z 366.998,A -85,B 0,C 180,E1 -14708.414,E2 -14708.414} C_VEL
LIN {X 0,Y 331.974,Z 366.678,A -85,B 0,C 180,E1 -14710.349,E2 -14710.349} C_VEL
LIN {X 0,Y 332.077,Z 366.211,A -85,B 0,C 180,E1 -14711.158,E2 -14711.158} C_VEL
LIN {X 0,Y 331.534,Z 365.5,A -85,B 0,C 180,E1 -14712.167,E2 -14712.167} C_VEL
LIN {X 0,Y 328.999,Z 363.859,A -85,B 0,C 180,E1 -14713.812,E2 -14713.812} C_VEL
LIN {X 0,Y 326.935,Z 362.131,A -85,B 0,C 180,E1 -14715.123,E2 -14715.123} C_VEL
LIN {X 0,Y 326.201,Z 360.381,A -85,B 0,C 180,E1 -14716.109,E2 -14716.109} C_VEL
LIN {X 0,Y 326.223,Z 359.692,A -85,B 0,C 180,E1 -14716.434,E2 -14716.434} C_VEL
LIN {X 0,Y 326.976,Z 355.432,A -85,B 0,C 180,E1 -14718.218,E2 -14718.218} C_VEL
LIN {X 0,Y 327.796,Z 350.162,A -85,B 0,C 180,E1 -14719.97,E2 -14719.97} C_VEL
LIN {X 0,Y 328.982,Z 343.6,A -85,B 0,C 180,E1 -14721.72,E2 -14721.72} C_VEL
LIN {X 0,Y 330.232,Z 335.704,A -85,B 0,C 180,E1 -14723.424,E2 -14723.424} C_VEL
LIN {X 0,Y 331.764,Z 325.951,A -85,B 0,C 180,E1 -14725.114,E2 -14725.114} C_VEL
LIN {X 0,Y 333.248,Z 315.462,A -85,B 0,C 180,E1 -14726.568,E2 -14726.568} C_VEL
LIN {X 0,Y 334.711,Z 304.013,A -85,B 0,C 180,E1 -14727.81,E2 -14727.81} C_VEL
LIN {X 0,Y 335.925,Z 292.102,A -85,B 0,C 180,E1 -14728.822,E2 -14728.822} C_VEL
LIN {X 0,Y 336.77,Z 280.612,A -85,B 0,C 180,E1 -14729.565,E2 -14729.565} C_VEL
LIN {X 0,Y 337.446,Z 267.814,A -85,B 0,C 180,E1 -14730.14,E2 -14730.14} C_VEL
LIN {X 0,Y 338.127,Z 248.415,A -85,B 0,C 180,E1 -14730.642,E2 -14730.642} C_VEL
LIN {X 0,Y 340.006,Z 185.538,A -85,B 0,C 180,E1 -14732.096,E2 -14732.096} C_VEL
LIN {X 0,Y 334.166,Z 171.112,A -85,B 0,C 180,E1 -14733.033,E2 -14733.033} C_VEL
LIN {X 0,Y 327.962,Z 157.901,A -85,B 0,C 180,E1 -14734.035,E2 -14734.035} C_VEL
LIN {X 0,Y 326.686,Z 152.797,A -85,B 0,C 180,E1 -14735.79,E2 -14735.79} C_VEL
LIN {X 0,Y 326.634,Z 152.8,A -85,B 0,C 180,E1 -14739.864,E2 -14739.864} C_VEL
LIN {X 0,Y 326.667,Z 152.793,A -85,B 0,C 180,E1 -14742.471,E2 -14742.471} C_VEL
LIN {X 0,Y 326.763,Z 152.785,A -85,B 0,C 180,E1 -14746.316,E2 -14746.316} C_VEL
LIN {X 0,Y 326.787,Z 152.779,A -85,B 0,C 180,E1 -14750.094,E2 -14750.094} C_VEL
LIN {X 0,Y 326.947,Z 152.762,A -85,B 0,C 180,E1 -14753.831,E2 -14753.831} C_VEL
LIN {X 0,Y 327.014,Z 152.752,A -85,B 0,C 180,E1 -14757.537,E2 -14757.537} C_VEL
LIN {X 0,Y 327.033,Z 152.748,A -85,B 0,C 180,E1 -14761.232,E2 -14761.232} C_VEL
LIN {X 0,Y 326.743,Z 152.777,A -85,B 0,C 180,E1 -14763.7,E2 -14763.7} C_VEL
LIN {X 0,Y 326.948,Z 152.751,A -85,B 0,C 180,E1 -14766.171,E2 -14766.171} C_VEL
LIN {X 0,Y 326.784,Z 152.774,A -85,B 0,C 180,E1 -14769.908,E2 -14769.908} C_VEL
LIN {X 0,Y 326.727,Z 152.784,A -85,B 0,C 180,E1 -14773.687,E2 -14773.687} C_VEL
LIN {X 0,Y 326.621,Z 152.801,A -85,B 0,C 180,E1 -14777.533,E2 -14777.533} C_VEL
LIN {X 0,Y 326.587,Z 152.798,A -85,B 0,C 180,E1 -14780.14,E2 -14780.14} C_VEL
LIN {X 0,Y 326.578,Z 152.802,A -85,B 0,C 180,E1 -14782.791,E2 -14782.791} C_VEL
LIN {X 0,Y 326.599,Z 152.799,A -85,B 0,C 180,E1 -14786.866,E2 -14786.866} C_VEL
LIN {X 0,Y 326.576,Z 152.799,A -85,B 0,C 180,E1 -14791.098,E2 -14791.098} C_VEL
LIN {X 0,Y 326.612,Z 152.799,A -85,B 0,C 180,E1 -14794.02,E2 -14794.02} C_VEL
LIN {X 0,Y 326.628,Z 152.798,A -85,B 0,C 180,E1 -14797.237,E2 -14797.237} C_VEL
LIN {X 0,Y 326.549,Z 152.805,A -85,B 0,C 180,E1 -14801.124,E2 -14801.124} C_VEL
LIN {X 0,Y 326.565,Z 152.806,A -85,B 0,C 180,E1 -14803.526,E2 -14803.526} C_VEL
LIN {X 0,Y 326.578,Z 152.808,A -85,B 0,C 180,E1 -14807.029,E2 -14807.029} C_VEL
LIN {X 0,Y 326.587,Z 152.806,A -85,B 0,C 180,E1 -14811.385,E2 -14811.385} C_VEL
LIN {X 0,Y 326.643,Z 152.799,A -85,B 0,C 180,E1 -14815.237,E2 -14815.237} C_VEL
LIN {X 0,Y 326.658,Z 152.986,A -85,B 0,C 180,E1 -14815.986,E2 -14815.986} C_VEL
LIN {X 0,Y 329.593,Z 164.688,A -85,B 0,C 180,E1 -14819.573,E2 -14819.573} C_VEL
LIN {X 0,Y 331.924,Z 175.995,A -85,B 0,C 180,E1 -14822.785,E2 -14822.785} C_VEL
LIN {X 0,Y 331.975,Z 179.164,A -85,B 0,C 180,E1 -14823.603,E2 -14823.603} C_VEL
LIN {X 0,Y 331.589,Z 182.369,A -85,B 0,C 180,E1 -14824.382,E2 -14824.382} C_VEL
LIN {X 0,Y 336.467,Z 207.352,A -85,B 0,C 180,E1 -14825.515,E2 -14825.515} C_VEL
LIN {X 0,Y 338.891,Z 224.854,A -85,B 0,C 180,E1 -14826.184,E2 -14826.184} C_VEL
LIN {X 0,Y 337.096,Z 292.148,A -85,B 0,C 180,E1 -14827.779,E2 -14827.779} C_VEL
LIN {X 0,Y 336.196,Z 305.923,A -85,B 0,C 180,E1 -14828.339,E2 -14828.339} C_VEL
LIN {X 0,Y 335.03,Z 317.629,A -85,B 0,C 180,E1 -14829.027,E2 -14829.027} C_VEL
LIN {X 0,Y 333.816,Z 327.994,A -85,B 0,C 180,E1 -14829.833,E2 -14829.833} C_VEL
LIN {X 0,Y 332.257,Z 339.855,A -85,B 0,C 180,E1 -14831.021,E2 -14831.021} C_VEL
LIN {X 0,Y 330.644,Z 350.499,A -85,B 0,C 180,E1 -14832.368,E2 -14832.368} C_VEL
LIN {X 0,Y 329.263,Z 360.133,A -85,B 0,C 180,E1 -14833.889,E2 -14833.889} C_VEL
LIN {X 0,Y 327.896,Z 369.467,A -85,B 0,C 180,E1 -14835.73,E2 -14835.73} C_VEL
LIN {X 0,Y 326.66,Z 377,A -85,B 0,C 180,E1 -14837.575,E2 -14837.575} C_VEL
LIN {X 0,Y 325.85,Z 383.072,A -85,B 0,C 180,E1 -14839.435,E2 -14839.435} C_VEL
LIN {X 0,Y 325.324,Z 387.889,A -85,B 0,C 180,E1 -14841.302,E2 -14841.302} C_VEL
LIN {X 0,Y 324.996,Z 391.586,A -85,B 0,C 180,E1 -14843.169,E2 -14843.169} C_VEL
LIN {X 0,Y 324.887,Z 394.265,A -85,B 0,C 180,E1 -14845.035,E2 -14845.035} C_VEL
LIN {X 0,Y 324.914,Z 395.543,A -85,B 0,C 180,E1 -14846.279,E2 -14846.279} C_VEL
LIN {X 0,Y 324.897,Z 396.367,A -85,B 0,C 180,E1 -14847.52,E2 -14847.52} C_VEL
LIN {X 0,Y 324.965,Z 396.787,A -85,B 0,C 180,E1 -14848.76,E2 -14848.76} C_VEL
LIN {X 0,Y 325.043,Z 396.813,A -85,B 0,C 180,E1 -14849.999,E2 -14849.999} C_VEL
LIN {X 0,Y 324.973,Z 396.432,A -85,B 0,C 180,E1 -14851.238,E2 -14851.238} C_VEL
LIN {X 0,Y 324.912,Z 395.602,A -85,B 0,C 180,E1 -14852.479,E2 -14852.479} C_VEL
LIN {X 0,Y 324.945,Z 394.355,A -85,B 0,C 180,E1 -14853.72,E2 -14853.72} C_VEL
LIN {X 0,Y 324.933,Z 391.36,A -85,B 0,C 180,E1 -14855.762,E2 -14855.762} C_VEL
LIN {X 0,Y 325.104,Z 387.93,A -85,B 0,C 180,E1 -14857.452,E2 -14857.452} C_VEL
LIN {X 0,Y 325.416,Z 383.034,A -85,B 0,C 180,E1 -14859.321,E2 -14859.321} C_VEL
LIN {X 0,Y 325.916,Z 376.835,A -85,B 0,C 180,E1 -14861.19,E2 -14861.19} C_VEL
LIN {X 0,Y 326.854,Z 369.125,A -85,B 0,C 180,E1 -14863.047,E2 -14863.047} C_VEL
LIN {X 0,Y 327.782,Z 361.208,A -85,B 0,C 180,E1 -14864.591,E2 -14864.591} C_VEL
LIN {X 0,Y 328.794,Z 351.513,A -85,B 0,C 180,E1 -14866.133,E2 -14866.133} C_VEL
LIN {X 0,Y 329.781,Z 342.07,A -85,B 0,C 180,E1 -14867.358,E2 -14867.358} C_VEL
LIN {X 0,Y 331.081,Z 330.422,A -85,B 0,C 180,E1 -14868.566,E2 -14868.566} C_VEL
LIN {X 0,Y 332.234,Z 318.096,A -85,B 0,C 180,E1 -14869.541,E2 -14869.541} C_VEL
LIN {X 0,Y 333.284,Z 304.493,A -85,B 0,C 180,E1 -14870.32,E2 -14870.32} C_VEL
LIN {X 0,Y 333.861,Z 291.674,A -85,B 0,C 180,E1 -14870.807,E2 -14870.807} C_VEL
LIN {X 0,Y 335.379,Z 224.394,A -85,B 0,C 180,E1 -14872.353,E2 -14872.353} C_VEL
LIN {X 0,Y 329.749,Z 184.379,A -85,B 0,C 180,E1 -14873.693,E2 -14873.693} C_VEL
LIN {X 0,Y 330.894,Z 174.188,A -85,B 0,C 180,E1 -14876.149,E2 -14876.149} C_VEL
LIN {X 0,Y 328.935,Z 163.147,A -85,B 0,C 180,E1 -14879.067,E2 -14879.067} C_VEL
LIN {X 0,Y 326.636,Z 152.8,A -85,B 0,C 180,E1 -14881.948,E2 -14881.948} C_VEL
LIN {X 0,Y 326.613,Z 152.8,A -85,B 0,C 180,E1 -14885.519,E2 -14885.519} C_VEL
LIN {X 0,Y 326.612,Z 152.799,A -85,B 0,C 180,E1 -14889.226,E2 -14889.226} C_VEL
LIN {X 0,Y 326.576,Z 152.803,A -85,B 0,C 180,E1 -14892.971,E2 -14892.971} C_VEL
LIN {X 0,Y 326.576,Z 152.803,A -85,B 0,C 180,E1 -14897.027,E2 -14897.027} C_VEL
LIN {X 0,Y 326.611,Z 152.798,A -85,B 0,C 180,E1 -14900.772,E2 -14900.772} C_VEL
LIN {X 0,Y 326.611,Z 152.798,A -85,B 0,C 180,E1 -14904.479,E2 -14904.479} C_VEL
LIN {X 0,Y 326.607,Z 152.804,A -85,B 0,C 180,E1 -14907.455,E2 -14907.455} C_VEL
LIN {X 0,Y 326.659,Z 152.791,A -85,B 0,C 180,E1 -14910.34,E2 -14910.34} C_VEL
LIN {X 0,Y 326.689,Z 152.788,A -85,B 0,C 180,E1 -14914.515,E2 -14914.515} C_VEL
LIN {X 0,Y 326.643,Z 152.794,A -85,B 0,C 180,E1 -14918.544,E2 -14918.544} C_VEL
LIN {X 0,Y 326.705,Z 152.791,A -85,B 0,C 180,E1 -14921.174,E2 -14921.174} C_VEL
LIN {X 0,Y 326.761,Z 152.782,A -85,B 0,C 180,E1 -14925.432,E2 -14925.432} C_VEL
LIN {X 0,Y 326.768,Z 152.782,A -85,B 0,C 180,E1 -14928.838,E2 -14928.838} C_VEL
LIN {X 0,Y 326.964,Z 152.755,A -85,B 0,C 180,E1 -14932.589,E2 -14932.589} C_VEL
LIN {X 0,Y 326.775,Z 152.782,A -85,B 0,C 180,E1 -14935.064,E2 -14935.064} C_VEL
LIN {X 0,Y 327.046,Z 152.744,A -85,B 0,C 180,E1 -14937.536,E2 -14937.536} C_VEL
LIN {X 0,Y 327.215,Z 152.722,A -85,B 0,C 180,E1 -14939.999,E2 -14939.999} C_VEL
LIN {X 0,Y 327.045,Z 152.746,A -85,B 0,C 180,E1 -14942.463,E2 -14942.463} C_VEL
LIN {X 0,Y 326.962,Z 152.753,A -85,B 0,C 180,E1 -14946.59,E2 -14946.59} C_VEL
LIN {X 0,Y 326.911,Z 152.766,A -85,B 0,C 180,E1 -14948.654,E2 -14948.654} C_VEL
LIN {X 0,Y 326.732,Z 152.786,A -85,B 0,C 180,E1 -14952.421,E2 -14952.421} C_VEL
LIN {X 0,Y 326.75,Z 152.782,A -85,B 0,C 180,E1 -14954.957,E2 -14954.957} C_VEL
LIN {X 0,Y 326.73,Z 152.785,A -85,B 0,C 180,E1 -14958.838,E2 -14958.838} C_VEL
LIN {X 0,Y 326.619,Z 152.798,A -85,B 0,C 180,E1 -14962.787,E2 -14962.787} C_VEL
LIN {X 0,Y 326.686,Z 152.787,A -85,B 0,C 180,E1 -14965.483,E2 -14965.483} C_VEL
LIN {X 0,Y 326.656,Z 152.793,A -85,B 0,C 180,E1 -14969.659,E2 -14969.659} C_VEL
LIN {X 0,Y 326.603,Z 152.803,A -85,B 0,C 180,E1 -14974.019,E2 -14974.019} C_VEL
LIN {X 0,Y 326.625,Z 152.795,A -85,B 0,C 180,E1 -14977.239,E2 -14977.239} C_VEL
LIN {X 0,Y 326.63,Z 152.799,A -85,B 0,C 180,E1 -14980.202,E2 -14980.202} C_VEL
LIN {X 0,Y 326.654,Z 152.794,A -85,B 0,C 180,E1 -14983.509,E2 -14983.509} C_VEL
LIN {X 0,Y 326.646,Z 152.793,A -85,B 0,C 180,E1 -14987.014,E2 -14987.014} C_VEL
LIN {X 0,Y 326.64,Z 152.794,A -85,B 0,C 180,E1 -14990.766,E2 -14990.766} C_VEL
LIN {X 0,Y 326.607,Z 152.798,A -85,B 0,C 180,E1 -14994.481,E2 -14994.481} C_VEL
LIN {X 0,Y 326.604,Z 152.802,A -85,B 0,C 180,E1 -14997.456,E2 -14997.456} C_VEL
LIN {X 0,Y 326.655,Z 152.793,A -85,B 0,C 180,E1 -15000.341,E2 -15000.341} C_VEL
LIN {X 0,Y 326.685,Z 152.789,A -85,B 0,C 180,E1 -15004.517,E2 -15004.517} C_VEL
LIN {X 0,Y 326.642,Z 152.794,A -85,B 0,C 180,E1 -15008.546,E2 -15008.546} C_VEL
LIN {X 0,Y 326.739,Z 152.786,A -85,B 0,C 180,E1 -15011.178,E2 -15011.178} C_VEL
LIN {X 0,Y 326.758,Z 152.784,A -85,B 0,C 180,E1 -15015.433,E2 -15015.433} C_VEL
LIN {X 0,Y 326.766,Z 152.781,A -85,B 0,C 180,E1 -15018.84,E2 -15018.84} C_VEL
LIN {X 0,Y 326.976,Z 152.754,A -85,B 0,C 180,E1 -15022.591,E2 -15022.591} C_VEL
LIN {X 0,Y 326.776,Z 152.783,A -85,B 0,C 180,E1 -15025.066,E2 -15025.066} C_VEL
LIN {X 0,Y 327.044,Z 152.745,A -85,B 0,C 180,E1 -15027.537,E2 -15027.537} C_VEL
LIN {X 0,Y 327.195,Z 152.725,A -85,B 0,C 180,E1 -15030.001,E2 -15030.001} C_VEL
LIN {X 0,Y 327.045,Z 152.745,A -85,B 0,C 180,E1 -15032.464,E2 -15032.464} C_VEL
LIN {X 0,Y 326.994,Z 152.751,A -85,B 0,C 180,E1 -15036.17,E2 -15036.17} C_VEL
LIN {X 0,Y 326.911,Z 152.765,A -85,B 0,C 180,E1 -15038.656,E2 -15038.656} C_VEL
LIN {X 0,Y 326.782,Z 152.797,A -85,B 0,C 180,E1 -15043.21,E2 -15043.21} C_VEL
LIN {X 0,Y 327.527,Z 156.351,A -85,B 0,C 180,E1 -15044.259,E2 -15044.259} C_VEL
LIN {X 0,Y 335.15,Z 178.287,A -85,B 0,C 180,E1 -15045.292,E2 -15045.292} C_VEL
LIN {X 0,Y 336.15,Z 184.303,A -85,B 0,C 180,E1 -15045.5,E2 -15045.5} C_VEL
LIN {X 0,Y 334.172,Z 264.196,A -85,B 0,C 180,E1 -15047.341,E2 -15047.341} C_VEL
LIN {X 0,Y 333.493,Z 277.919,A -85,B 0,C 180,E1 -15047.912,E2 -15047.912} C_VEL
LIN {X 0,Y 332.787,Z 290.674,A -85,B 0,C 180,E1 -15048.708,E2 -15048.708} C_VEL
LIN {X 0,Y 331.963,Z 301.835,A -85,B 0,C 180,E1 -15049.64,E2 -15049.64} C_VEL
LIN {X 0,Y 330.839,Z 313.056,A -85,B 0,C 180,E1 -15050.824,E2 -15050.824} C_VEL
LIN {X 0,Y 329.663,Z 323.711,A -85,B 0,C 180,E1 -15052.236,E2 -15052.236} C_VEL
LIN {X 0,Y 328.63,Z 333.018,A -85,B 0,C 180,E1 -15053.78,E2 -15053.78} C_VEL
LIN {X 0,Y 327.543,Z 342.28,A -85,B 0,C 180,E1 -15055.688,E2 -15055.688} C_VEL
LIN {X 0,Y 326.747,Z 349.087,A -85,B 0,C 180,E1 -15057.441,E2 -15057.441} C_VEL
LIN {X 0,Y 326.172,Z 354.013,A -85,B 0,C 180,E1 -15059.001,E2 -15059.001} C_VEL
LIN {X 0,Y 325.57,Z 359.488,A -85,B 0,C 180,E1 -15061.205,E2 -15061.205} C_VEL
LIN {X 0,Y 325.147,Z 363.473,A -85,B 0,C 180,E1 -15063.449,E2 -15063.449} C_VEL
LIN {X 0,Y 324.797,Z 366.099,A -85,B 0,C 180,E1 -15065.749,E2 -15065.749} C_VEL
LIN {X 0,Y 324.752,Z 367.019,A -85,B 0,C 180,E1 -15067.298,E2 -15067.298} C_VEL
LIN {X 0,Y 324.802,Z 367.354,A -85,B 0,C 180,E1 -15068.867,E2 -15068.867} C_VEL
LIN {X 0,Y 324.976,Z 366.601,A -85,B 0,C 180,E1 -15071.189,E2 -15071.189} C_VEL
LIN {X 0,Y 325.23,Z 365.416,A -85,B 0,C 180,E1 -15072.718,E2 -15072.718} C_VEL
LIN {X 0,Y 325.709,Z 363.017,A -85,B 0,C 180,E1 -15074.598,E2 -15074.598} C_VEL
LIN {X 0,Y 326.223,Z 359.692,A -85,B 0,C 180,E1 -15076.434,E2 -15076.434} C_VEL
LIN {X 0,Y 325.907,Z 357.619,A -85,B 0,C 180,E1 -15077.401,E2 -15077.401} C_VEL
LIN {X 0,Y 323.758,Z 353.878,A -85,B 0,C 180,E1 -15078.981,E2 -15078.981} C_VEL
LIN {X 0,Y 321.766,Z 349.605,A -85,B 0,C 180,E1 -15080.529,E2 -15080.529} C_VEL
LIN {X 0,Y 321.695,Z 346.527,A -85,B 0,C 180,E1 -15081.429,E2 -15081.429} C_VEL
LIN {X 0,Y 323.07,Z 338.427,A -85,B 0,C 180,E1 -15083.344,E2 -15083.344} C_VEL
LIN {X 0,Y 324.687,Z 329.113,A -85,B 0,C 180,E1 -15085.097,E2 -15085.097} C_VEL
LIN {X 0,Y 326.267,Z 318.584,A -85,B 0,C 180,E1 -15086.669,E2 -15086.669} C_VEL
LIN {X 0,Y 327.724,Z 308.411,A -85,B 0,C 180,E1 -15087.88,E2 -15087.88} C_VEL
LIN {X 0,Y 328.917,Z 297.841,A -85,B 0,C 180,E1 -15088.896,E2 -15088.896} C_VEL
LIN {X 0,Y 329.995,Z 286.356,A -85,B 0,C 180,E1 -15089.754,E2 -15089.754} C_VEL
LIN {X 0,Y 330.788,Z 274.563,A -85,B 0,C 180,E1 -15090.402,E2 -15090.402} C_VEL
LIN {X 0,Y 331.365,Z 262.985,A -85,B 0,C 180,E1 -15090.832,E2 -15090.832} C_VEL
LIN {X 0,Y 333.682,Z 187.02,A -85,B 0,C 180,E1 -15092.652,E2 -15092.652} C_VEL
LIN {X 0,Y 327.795,Z 172.88,A -85,B 0,C 180,E1 -15093.619,E2 -15093.619} C_VEL
LIN {X 0,Y 322.099,Z 161.068,A -85,B 0,C 180,E1 -15094.561,E2 -15094.561} C_VEL
LIN {X 0,Y 320.829,Z 158.319,A -85,B 0,C 180,E1 -15094.8,E2 -15094.8} C_VEL
LIN {X 0,Y 319.589,Z 153.681,A -85,B 0,C 180,E1 -15096.425,E2 -15096.425} C_VEL
LIN {X 0,Y 319.643,Z 153.669,A -85,B 0,C 180,E1 -15100.989,E2 -15100.989} C_VEL
LIN {X 0,Y 319.716,Z 153.664,A -85,B 0,C 180,E1 -15105.29,E2 -15105.29} C_VEL
LIN {X 0,Y 319.719,Z 153.664,A -85,B 0,C 180,E1 -15108.59,E2 -15108.59} C_VEL
LIN {X 0,Y 319.857,Z 153.642,A -85,B 0,C 180,E1 -15112.425,E2 -15112.425} C_VEL
LIN {X 0,Y 319.723,Z 153.658,A -85,B 0,C 180,E1 -15114.956,E2 -15114.956} C_VEL
LIN {X 0,Y 319.96,Z 153.63,A -85,B 0,C 180,E1 -15117.483,E2 -15117.483} C_VEL
LIN {X 0,Y 320.003,Z 153.624,A -85,B 0,C 180,E1 -15121.259,E2 -15121.259} C_VEL
LIN {X 0,Y 319.721,Z 153.658,A -85,B 0,C 180,E1 -15125.045,E2 -15125.045} C_VEL
LIN {X 0,Y 319.859,Z 153.632,A -85,B 0,C 180,E1 -15127.576,E2 -15127.576} C_VEL
LIN {X 0,Y 319.709,Z 153.649,A -85,B 0,C 180,E1 -15131.412,E2 -15131.412} C_VEL
LIN {X 0,Y 319.654,Z 153.658,A -85,B 0,C 180,E1 -15134.668,E2 -15134.668} C_VEL
LIN {X 0,Y 319.602,Z 153.666,A -85,B 0,C 180,E1 -15138.99,E2 -15138.99} C_VEL
LIN {X 0,Y 319.524,Z 153.676,A -85,B 0,C 180,E1 -15143.324,E2 -15143.324} C_VEL
LIN {X 0,Y 319.553,Z 153.679,A -85,B 0,C 180,E1 -15146.096,E2 -15146.096} C_VEL
LIN {X 0,Y 319.529,Z 153.68,A -85,B 0,C 180,E1 -15148.94,E2 -15148.94} C_VEL
LIN {X 0,Y 319.528,Z 153.676,A -85,B 0,C 180,E1 -15151.863,E2 -15151.863} C_VEL
LIN {X 0,Y 319.584,Z 153.671,A -85,B 0,C 180,E1 -15155.543,E2 -15155.543} C_VEL
LIN {X 0,Y 319.533,Z 153.683,A -85,B 0,C 180,E1 -15159.662,E2 -15159.662} C_VEL
LIN {X 0,Y 319.525,Z 153.683,A -85,B 0,C 180,E1 -15163.46,E2 -15163.46} C_VEL
LIN {X 0,Y 319.557,Z 153.683,A -85,B 0,C 180,E1 -15167.016,E2 -15167.016} C_VEL
LIN {X 0,Y 319.519,Z 153.686,A -85,B 0,C 180,E1 -15170.366,E2 -15170.366} C_VEL
LIN {X 0,Y 319.561,Z 153.68,A -85,B 0,C 180,E1 -15173.572,E2 -15173.572} C_VEL
LIN {X 0,Y 319.628,Z 153.871,A -85,B 0,C 180,E1 -15175.319,E2 -15175.319} C_VEL
LIN {X 0,Y 322.274,Z 164.222,A -85,B 0,C 180,E1 -15178.631,E2 -15178.631} C_VEL
LIN {X 0,Y 324.159,Z 172.882,A -85,B 0,C 180,E1 -15181.212,E2 -15181.212} C_VEL
LIN {X 0,Y 325.296,Z 179.235,A -85,B 0,C 180,E1 -15183.018,E2 -15183.018} C_VEL
LIN {X 0,Y 325.008,Z 182.122,A -85,B 0,C 180,E1 -15183.712,E2 -15183.712} C_VEL
LIN {X 0,Y 329.491,Z 204.277,A -85,B 0,C 180,E1 -15184.771,E2 -15184.771} C_VEL
LIN {X 0,Y 332.529,Z 225.293,A -85,B 0,C 180,E1 -15185.627,E2 -15185.627} C_VEL
LIN {X 0,Y 330.953,Z 286.825,A -85,B 0,C 180,E1 -15187.107,E2 -15187.107} C_VEL
LIN {X 0,Y 330.115,Z 300.951,A -85,B 0,C 180,E1 -15187.59,E2 -15187.59} C_VEL
LIN {X 0,Y 328.899,Z 313.921,A -85,B 0,C 180,E1 -15188.287,E2 -15188.287} C_VEL
LIN {X 0,Y 327.35,Z 326.755,A -85,B 0,C 180,E1 -15189.252,E2 -15189.252} C_VEL
LIN {X 0,Y 325.942,Z 337.496,A -85,B 0,C 180,E1 -15190.311,E2 -15190.311} C_VEL
LIN {X 0,Y 324.238,Z 348.532,A -85,B 0,C 180,E1 -15191.681,E2 -15191.681} C_VEL
LIN {X 0,Y 322.681,Z 358.434,A -85,B 0,C 180,E1 -15193.226,E2 -15193.226} C_VEL
LIN {X 0,Y 321.381,Z 366.588,A -85,B 0,C 180,E1 -15194.786,E2 -15194.786} C_VEL
LIN {X 0,Y 320.136,Z 374.626,A -85,B 0,C 180,E1 -15196.672,E2 -15196.672} C_VEL
LIN {X 0,Y 319.057,Z 381.071,A -85,B 0,C 180,E1 -15198.565,E2 -15198.565} C_VEL
LIN {X 0,Y 318.429,Z 386.235,A -85,B 0,C 180,E1 -15200.471,E2 -15200.471} C_VEL
LIN {X 0,Y 318.017,Z 390.26,A -85,B 0,C 180,E1 -15202.38,E2 -15202.38} C_VEL
LIN {X 0,Y 317.831,Z 393.27,A -85,B 0,C 180,E1 -15204.307,E2 -15204.307} C_VEL
LIN {X 0,Y 317.819,Z 395.267,A -85,B 0,C 180,E1 -15206.195,E2 -15206.195} C_VEL
LIN {X 0,Y 317.815,Z 396.065,A -85,B 0,C 180,E1 -15207.464,E2 -15207.464} C_VEL
LIN {X 0,Y 317.869,Z 396.468,A -85,B 0,C 180,E1 -15208.732,E2 -15208.732} C_VEL
LIN {X 0,Y 317.95,Z 396.477,A -85,B 0,C 180,E1 -15209.999,E2 -15209.999} C_VEL
LIN {X 0,Y 317.877,Z 396.069,A -85,B 0,C 180,E1 -15211.266,E2 -15211.266} C_VEL
LIN {X 0,Y 317.829,Z 395.21,A -85,B 0,C 180,E1 -15212.534,E2 -15212.534} C_VEL
LIN {X 0,Y 317.871,Z 393.945,A -85,B 0,C 180,E1 -15213.802,E2 -15213.802} C_VEL
LIN {X 0,Y 317.851,Z 391.183,A -85,B 0,C 180,E1 -15215.729,E2 -15215.729} C_VEL
LIN {X 0,Y 318.025,Z 387.432,A -85,B 0,C 180,E1 -15217.619,E2 -15217.619} C_VEL
LIN {X 0,Y 318.36,Z 382.488,A -85,B 0,C 180,E1 -15219.529,E2 -15219.529} C_VEL
LIN {X 0,Y 318.904,Z 376.236,A -85,B 0,C 180,E1 -15221.439,E2 -15221.439} C_VEL
LIN {X 0,Y 319.9,Z 368.444,A -85,B 0,C 180,E1 -15223.336,E2 -15223.336} C_VEL
LIN {X 0,Y 320.849,Z 360.438,A -85,B 0,C 180,E1 -15224.914,E2 -15224.914} C_VEL
LIN {X 0,Y 321.909,Z 350.652,A -85,B 0,C 180,E1 -15226.488,E2 -15226.488} C_VEL
LIN {X 0,Y 323.13,Z 339.799,A -85,B 0,C 180,E1 -15227.891,E2 -15227.891} C_VEL
LIN {X 0,Y 324.304,Z 329.274,A -85,B 0,C 180,E1 -15228.969,E2 -15228.969} C_VEL
LIN {X 0,Y 325.511,Z 316.65,A -85,B 0,C 180,E1 -15229.962,E2 -15229.962} C_VEL
LIN {X 0,Y 326.528,Z 303.411,A -85,B 0,C 180,E1 -15230.719,E2 -15230.719} C_VEL
LIN {X 0,Y 327.185,Z 289.959,A -85,B 0,C 180,E1 -15231.21,E2 -15231.21} C_VEL
LIN {X 0,Y 328.632,Z 224.937,A -85,B 0,C 180,E1 -15232.737,E2 -15232.737} C_VEL
LIN {X 0,Y 322.903,Z 184.097,A -85,B 0,C 180,E1 -15234.14,E2 -15234.14} C_VEL
LIN {X 0,Y 323.882,Z 174.898,A -85,B 0,C 180,E1 -15236.412,E2 -15236.412} C_VEL
LIN {X 0,Y 321.999,Z 164.634,A -85,B 0,C 180,E1 -15239.184,E2 -15239.184} C_VEL
LIN {X 0,Y 319.575,Z 153.679,A -85,B 0,C 180,E1 -15242.321,E2 -15242.321} C_VEL
LIN {X 0,Y 319.559,Z 153.678,A -85,B 0,C 180,E1 -15246.427,E2 -15246.427} C_VEL
LIN {X 0,Y 319.559,Z 153.68,A -85,B 0,C 180,E1 -15249.668,E2 -15249.668} C_VEL
LIN {X 0,Y 319.521,Z 153.684,A -85,B 0,C 180,E1 -15253.46,E2 -15253.46} C_VEL
LIN {X 0,Y 319.554,Z 153.678,A -85,B 0,C 180,E1 -15257.016,E2 -15257.016} C_VEL
LIN {X 0,Y 319.546,Z 153.678,A -85,B 0,C 180,E1 -15260.37,E2 -15260.37} C_VEL
LIN {X 0,Y 319.558,Z 153.682,A -85,B 0,C 180,E1 -15263.572,E2 -15263.572} C_VEL
LIN {X 0,Y 319.576,Z 153.674,A -85,B 0,C 180,E1 -15266.686,E2 -15266.686} C_VEL
LIN {X 0,Y 319.59,Z 153.676,A -85,B 0,C 180,E1 -15269.616,E2 -15269.616} C_VEL
LIN {X 0,Y 319.607,Z 153.67,A -85,B 0,C 180,E1 -15272.497,E2 -15272.497} C_VEL
LIN {X 0,Y 319.604,Z 153.676,A -85,B 0,C 180,E1 -15275.303,E2 -15275.303} C_VEL
LIN {X 0,Y 319.595,Z 153.672,A -85,B 0,C 180,E1 -15278.047,E2 -15278.047} C_VEL
LIN {X 0,Y 319.622,Z 153.668,A -85,B 0,C 180,E1 -15282.07,E2 -15282.07} C_VEL
LIN {X 0,Y 319.73,Z 153.655,A -85,B 0,C 180,E1 -15286.007,E2 -15286.007} C_VEL
LIN {X 0,Y 319.755,Z 153.652,A -85,B 0,C 180,E1 -15289.872,E2 -15289.872} C_VEL
LIN {X 0,Y 319.923,Z 153.631,A -85,B 0,C 180,E1 -15292.425,E2 -15292.425} C_VEL
LIN {X 0,Y 319.744,Z 153.658,A -85,B 0,C 180,E1 -15294.955,E2 -15294.955} C_VEL
LIN {X 0,Y 319.989,Z 153.624,A -85,B 0,C 180,E1 -15297.482,E2 -15297.482} C_VEL
LIN {X 0,Y 320.166,Z 153.6,A -85,B 0,C 180,E1 -15299.999,E2 -15299.999} C_VEL
LIN {X 0,Y 319.989,Z 153.624,A -85,B 0,C 180,E1 -15302.517,E2 -15302.517} C_VEL
LIN {X 0,Y 319.924,Z 153.63,A -85,B 0,C 180,E1 -15306.579,E2 -15306.579} C_VEL
LIN {X 0,Y 319.839,Z 153.645,A -85,B 0,C 180,E1 -15308.847,E2 -15308.847} C_VEL
LIN {X 0,Y 319.679,Z 153.664,A -85,B 0,C 180,E1 -15312.699,E2 -15312.699} C_VEL
LIN {X 0,Y 319.696,Z 153.658,A -85,B 0,C 180,E1 -15315.295,E2 -15315.295} C_VEL
LIN {X 0,Y 319.672,Z 153.662,A -85,B 0,C 180,E1 -15319.254,E2 -15319.254} C_VEL
LIN {X 0,Y 319.568,Z 153.674,A -85,B 0,C 180,E1 -15323.319,E2 -15323.319} C_VEL
LIN {X 0,Y 319.63,Z 153.669,A -85,B 0,C 180,E1 -15326.088,E2 -15326.088} C_VEL
LIN {X 0,Y 319.584,Z 153.673,A -85,B 0,C 180,E1 -15328.933,E2 -15328.933} C_VEL
LIN {X 0,Y 319.528,Z 153.682,A -85,B 0,C 180,E1 -15331.861,E2 -15331.861} C_VEL
LIN {X 0,Y 319.575,Z 153.674,A -85,B 0,C 180,E1 -15335.543,E2 -15335.543} C_VEL
LIN {X 0,Y 319.595,Z 153.675,A -85,B 0,C 180,E1 -15338.004,E2 -15338.004} C_VEL
LIN {X 0,Y 319.597,Z 153.673,A -85,B 0,C 180,E1 -15341.612,E2 -15341.612} C_VEL
LIN {X 0,Y 319.641,Z 153.666,A -85,B 0,C 180,E1 -15345.285,E2 -15345.285} C_VEL
LIN {X 0,Y 319.578,Z 153.674,A -85,B 0,C 180,E1 -15348.721,E2 -15348.721} C_VEL
LIN {X 0,Y 319.593,Z 153.673,A -85,B 0,C 180,E1 -15352.339,E2 -15352.339} C_VEL
LIN {X 0,Y 319.555,Z 153.677,A -85,B 0,C 180,E1 -15355.124,E2 -15355.124} C_VEL
LIN {X 0,Y 319.565,Z 153.677,A -85,B 0,C 180,E1 -15359.058,E2 -15359.058} C_VEL
LIN {X 0,Y 319.603,Z 153.671,A -85,B 0,C 180,E1 -15362.498,E2 -15362.498} C_VEL
LIN {X 0,Y 319.6,Z 153.675,A -85,B 0,C 180,E1 -15365.304,E2 -15365.304} C_VEL
LIN {X 0,Y 319.592,Z 153.673,A -85,B 0,C 180,E1 -15368.048,E2 -15368.048} C_VEL
LIN {X 0,Y 319.684,Z 153.663,A -85,B 0,C 180,E1 -15370.962,E2 -15370.962} C_VEL
LIN {X 0,Y 319.726,Z 153.661,A -85,B 0,C 180,E1 -15375.276,E2 -15375.276} C_VEL
LIN {X 0,Y 319.754,Z 153.653,A -85,B 0,C 180,E1 -15379.873,E2 -15379.873} C_VEL
LIN {X 0,Y 319.929,Z 153.631,A -85,B 0,C 180,E1 -15382.427,E2 -15382.427} C_VEL
LIN {X 0,Y 319.745,Z 153.658,A -85,B 0,C 180,E1 -15384.957,E2 -15384.957} C_VEL
LIN {X 0,Y 319.988,Z 153.625,A -85,B 0,C 180,E1 -15387.483,E2 -15387.483} C_VEL
LIN {X 0,Y 320.147,Z 153.603,A -85,B 0,C 180,E1 -15390.001,E2 -15390.001} C_VEL
LIN {X 0,Y 319.988,Z 153.625,A -85,B 0,C 180,E1 -15392.518,E2 -15392.518} C_VEL
LIN {X 0,Y 319.949,Z 153.629,A -85,B 0,C 180,E1 -15396.306,E2 -15396.306} C_VEL
LIN {X 0,Y 319.839,Z 153.647,A -85,B 0,C 180,E1 -15398.849,E2 -15398.849} C_VEL
LIN {X 0,Y 319.736,Z 153.865,A -85,B 0,C 180,E1 -15402.941,E2 -15402.941} C_VEL
LIN {X 0,Y 320.32,Z 156.509,A -85,B 0,C 180,E1 -15403.764,E2 -15403.764} C_VEL
LIN {X 0,Y 328.224,Z 178.885,A -85,B 0,C 180,E1 -15404.87,E2 -15404.87} C_VEL
LIN {X 0,Y 329.473,Z 185.283,A -85,B 0,C 180,E1 -15405.109,E2 -15405.109} C_VEL
LIN {X 0,Y 327.436,Z 264.237,A -85,B 0,C 180,E1 -15406.965,E2 -15406.965} C_VEL
LIN {X 0,Y 326.708,Z 278.32,A -85,B 0,C 180,E1 -15407.561,E2 -15407.561} C_VEL
LIN {X 0,Y 326.035,Z 290.035,A -85,B 0,C 180,E1 -15408.296,E2 -15408.296} C_VEL
LIN {X 0,Y 325.177,Z 301.404,A -85,B 0,C 180,E1 -15409.245,E2 -15409.245} C_VEL
LIN {X 0,Y 323.954,Z 313.397,A -85,B 0,C 180,E1 -15410.529,E2 -15410.529} C_VEL
LIN {X 0,Y 322.807,Z 323.521,A -85,B 0,C 180,E1 -15411.892,E2 -15411.892} C_VEL
LIN {X 0,Y 321.731,Z 332.813,A -85,B 0,C 180,E1 -15413.444,E2 -15413.444} C_VEL
LIN {X 0,Y 320.644,Z 341.781,A -85,B 0,C 180,E1 -15415.304,E2 -15415.304} C_VEL
LIN {X 0,Y 319.775,Z 348.884,A -85,B 0,C 180,E1 -15417.133,E2 -15417.133} C_VEL
LIN {X 0,Y 319.081,Z 354.655,A -85,B 0,C 180,E1 -15418.985,E2 -15418.985} C_VEL
LIN {X 0,Y 318.478,Z 360.107,A -85,B 0,C 180,E1 -15421.275,E2 -15421.275} C_VEL
LIN {X 0,Y 318.055,Z 363.965,A -85,B 0,C 180,E1 -15423.534,E2 -15423.534} C_VEL
LIN {X 0,Y 317.779,Z 365.811,A -85,B 0,C 180,E1 -15425.102,E2 -15425.102} C_VEL
LIN {X 0,Y 317.675,Z 367.288,A -85,B 0,C 180,E1 -15427.21,E2 -15427.21} C_VEL
LIN {X 0,Y 317.714,Z 367.656,A -85,B 0,C 180,E1 -15429.267,E2 -15429.267} C_VEL
LIN {X 0,Y 317.94,Z 366.835,A -85,B 0,C 180,E1 -15431.541,E2 -15431.541} C_VEL
LIN {X 0,Y 318.462,Z 364.42,A -85,B 0,C 180,E1 -15434.04,E2 -15434.04} C_VEL
LIN {X 0,Y 318.971,Z 361.708,A -85,B 0,C 180,E1 -15435.813,E2 -15435.813} C_VEL
LIN {X 0,Y 319.611,Z 358.038,A -85,B 0,C 180,E1 -15437.601,E2 -15437.601} C_VEL
LIN {X 0,Y 320.61,Z 352.319,A -85,B 0,C 180,E1 -15439.73,E2 -15439.73} C_VEL
LIN {X 0,Y 321.695,Z 346.527,A -85,B 0,C 180,E1 -15441.429,E2 -15441.429} C_VEL
LIN {X 0,Y 321.668,Z 343.258,A -85,B 0,C 180,E1 -15442.306,E2 -15442.306} C_VEL
LIN {X 0,Y 319.951,Z 337.724,A -85,B 0,C 180,E1 -15443.744,E2 -15443.744} C_VEL
LIN {X 0,Y 318.289,Z 331.629,A -85,B 0,C 180,E1 -15445.115,E2 -15445.115} C_VEL
LIN {X 0,Y 318.335,Z 327.483,A -85,B 0,C 180,E1 -15445.871,E2 -15445.871} C_VEL
LIN {X 0,Y 320.051,Z 316.664,A -85,B 0,C 180,E1 -15447.454,E2 -15447.454} C_VEL
LIN {X 0,Y 321.577,Z 306.149,A -85,B 0,C 180,E1 -15448.663,E2 -15448.663} C_VEL
LIN {X 0,Y 322.873,Z 294.932,A -85,B 0,C 180,E1 -15449.688,E2 -15449.688} C_VEL
LIN {X 0,Y 323.966,Z 281.746,A -85,B 0,C 180,E1 -15450.606,E2 -15450.606} C_VEL
LIN {X 0,Y 324.779,Z 268.359,A -85,B 0,C 180,E1 -15451.233,E2 -15451.233} C_VEL
LIN {X 0,Y 325.502,Z 248.828,A -85,B 0,C 180,E1 -15451.762,E2 -15451.762} C_VEL
LIN {X 0,Y 327.459,Z 188.863,A -85,B 0,C 180,E1 -15453.212,E2 -15453.212} C_VEL
LIN {X 0,Y 321.095,Z 173.753,A -85,B 0,C 180,E1 -15454.305,E2 -15454.305} C_VEL
LIN {X 0,Y 314.966,Z 161.502,A -85,B 0,C 180,E1 -15455.357,E2 -15455.357} C_VEL
LIN {X 0,Y 313.679,Z 158.762,A -85,B 0,C 180,E1 -15455.602,E2 -15455.602} C_VEL
LIN {X 0,Y 312.535,Z 154.559,A -85,B 0,C 180,E1 -15457.218,E2 -15457.218} C_VEL
LIN {X 0,Y 312.585,Z 154.549,A -85,B 0,C 180,E1 -15461.654,E2 -15461.654} C_VEL
LIN {X 0,Y 312.689,Z 154.539,A -85,B 0,C 180,E1 -15465.687,E2 -15465.687} C_VEL
LIN {X 0,Y 312.69,Z 154.534,A -85,B 0,C 180,E1 -15469.642,E2 -15469.642} C_VEL
LIN {X 0,Y 312.8,Z 154.521,A -85,B 0,C 180,E1 -15472.253,E2 -15472.253} C_VEL
LIN {X 0,Y 312.693,Z 154.534,A -85,B 0,C 180,E1 -15474.843,E2 -15474.843} C_VEL
LIN {X 0,Y 312.971,Z 154.493,A -85,B 0,C 180,E1 -15478.714,E2 -15478.714} C_VEL
LIN {X 0,Y 312.971,Z 154.5,A -85,B 0,C 180,E1 -15481.287,E2 -15481.287} C_VEL
LIN {X 0,Y 312.846,Z 154.505,A -85,B 0,C 180,E1 -15486.45,E2 -15486.45} C_VEL
LIN {X 0,Y 312.755,Z 154.525,A -85,B 0,C 180,E1 -15489.051,E2 -15489.051} C_VEL
LIN {X 0,Y 312.611,Z 154.542,A -85,B 0,C 180,E1 -15492.993,E2 -15492.993} C_VEL
LIN {X 0,Y 312.547,Z 154.542,A -85,B 0,C 180,E1 -15495.655,E2 -15495.655} C_VEL
LIN {X 0,Y 312.52,Z 154.547,A -85,B 0,C 180,E1 -15499.715,E2 -15499.715} C_VEL
LIN {X 0,Y 312.505,Z 154.554,A -85,B 0,C 180,E1 -15502.769,E2 -15502.769} C_VEL
LIN {X 0,Y 312.486,Z 154.557,A -85,B 0,C 180,E1 -15506.732,E2 -15506.732} C_VEL
LIN {X 0,Y 312.473,Z 154.562,A -85,B 0,C 180,E1 -15509.658,E2 -15509.658} C_VEL
LIN {X 0,Y 312.525,Z 154.555,A -85,B 0,C 180,E1 -15513.689,E2 -15513.689} C_VEL
LIN {X 0,Y 312.519,Z 154.554,A -85,B 0,C 180,E1 -15517.387,E2 -15517.387} C_VEL
LIN {X 0,Y 312.446,Z 154.564,A -85,B 0,C 180,E1 -15520.717,E2 -15520.717} C_VEL
LIN {X 0,Y 312.456,Z 154.563,A -85,B 0,C 180,E1 -15524.21,E2 -15524.21} C_VEL
LIN {X 0,Y 312.461,Z 154.569,A -85,B 0,C 180,E1 -15527.924,E2 -15527.924} C_VEL
LIN {X 0,Y 312.489,Z 154.562,A -85,B 0,C 180,E1 -15531.922,E2 -15531.922} C_VEL
LIN {X 0,Y 312.572,Z 154.635,A -85,B 0,C 180,E1 -15534.571,E2 -15534.571} C_VEL
LIN {X 0,Y 315.651,Z 166.673,A -85,B 0,C 180,E1 -15538.548,E2 -15538.548} C_VEL
LIN {X 0,Y 317.506,Z 175.438,A -85,B 0,C 180,E1 -15541.218,E2 -15541.218} C_VEL
LIN {X 0,Y 318.458,Z 181.33,A -85,B 0,C 180,E1 -15542.923,E2 -15542.923} C_VEL
LIN {X 0,Y 318.804,Z 183.408,A -85,B 0,C 180,E1 -15543.081,E2 -15543.081} C_VEL
LIN {X 0,Y 322.322,Z 200.242,A -85,B 0,C 180,E1 -15543.943,E2 -15543.943} C_VEL
LIN {X 0,Y 325.093,Z 216.935,A -85,B 0,C 180,E1 -15544.687,E2 -15544.687} C_VEL
LIN {X 0,Y 326.376,Z 227.672,A -85,B 0,C 180,E1 -15545.107,E2 -15545.107} C_VEL
LIN {X 0,Y 324.366,Z 291.393,A -85,B 0,C 180,E1 -15546.678,E2 -15546.678} C_VEL
LIN {X 0,Y 323.405,Z 305.302,A -85,B 0,C 180,E1 -15547.268,E2 -15547.268} C_VEL
LIN {X 0,Y 322.122,Z 316.954,A -85,B 0,C 180,E1 -15547.975,E2 -15547.975} C_VEL
LIN {X 0,Y 320.589,Z 328.925,A -85,B 0,C 180,E1 -15548.962,E2 -15548.962} C_VEL
LIN {X 0,Y 318.909,Z 340.43,A -85,B 0,C 180,E1 -15550.194,E2 -15550.194} C_VEL
LIN {X 0,Y 317.163,Z 350.869,A -85,B 0,C 180,E1 -15551.592,E2 -15551.592} C_VEL
LIN {X 0,Y 315.447,Z 361.176,A -85,B 0,C 180,E1 -15553.341,E2 -15553.341} C_VEL
LIN {X 0,Y 314.103,Z 369.449,A -85,B 0,C 180,E1 -15555.089,E2 -15555.089} C_VEL
LIN {X 0,Y 312.801,Z 376.859,A -85,B 0,C 180,E1 -15557.015,E2 -15557.015} C_VEL
LIN {X 0,Y 311.842,Z 382.823,A -85,B 0,C 180,E1 -15558.955,E2 -15558.955} C_VEL
LIN {X 0,Y 311.234,Z 387.544,A -85,B 0,C 180,E1 -15560.904,E2 -15560.904} C_VEL
LIN {X 0,Y 310.84,Z 391.16,A -85,B 0,C 180,E1 -15562.856,E2 -15562.856} C_VEL
LIN {X 0,Y 310.705,Z 393.765,A -85,B 0,C 180,E1 -15564.808,E2 -15564.808} C_VEL
LIN {X 0,Y 310.728,Z 394.985,A -85,B 0,C 180,E1 -15566.109,E2 -15566.109} C_VEL
LIN {X 0,Y 310.734,Z 395.764,A -85,B 0,C 180,E1 -15567.407,E2 -15567.407} C_VEL
LIN {X 0,Y 310.775,Z 396.15,A -85,B 0,C 180,E1 -15568.703,E2 -15568.703} C_VEL
LIN {X 0,Y 310.857,Z 396.141,A -85,B 0,C 180,E1 -15569.999,E2 -15569.999} C_VEL
LIN {X 0,Y 310.784,Z 395.7,A -85,B 0,C 180,E1 -15571.295,E2 -15571.295} C_VEL
LIN {X 0,Y 310.749,Z 394.82,A -85,B 0,C 180,E1 -15572.592,E2 -15572.592} C_VEL
LIN {X 0,Y 310.775,Z 393.533,A -85,B 0,C 180,E1 -15573.889,E2 -15573.889} C_VEL
LIN {X 0,Y 310.768,Z 391.008,A -85,B 0,C 180,E1 -15575.693,E2 -15575.693} C_VEL
LIN {X 0,Y 310.973,Z 386.936,A -85,B 0,C 180,E1 -15577.793,E2 -15577.793} C_VEL
LIN {X 0,Y 311.322,Z 381.943,A -85,B 0,C 180,E1 -15579.747,E2 -15579.747} C_VEL
LIN {X 0,Y 311.89,Z 375.635,A -85,B 0,C 180,E1 -15581.7,E2 -15581.7} C_VEL
LIN {X 0,Y 312.936,Z 367.751,A -85,B 0,C 180,E1 -15583.639,E2 -15583.639} C_VEL
LIN {X 0,Y 313.937,Z 359.669,A -85,B 0,C 180,E1 -15585.25,E2 -15585.25} C_VEL
LIN {X 0,Y 315.033,Z 349.789,A -85,B 0,C 180,E1 -15586.858,E2 -15586.858} C_VEL
LIN {X 0,Y 316.375,Z 338.811,A -85,B 0,C 180,E1 -15588.286,E2 -15588.286} C_VEL
LIN {X 0,Y 317.732,Z 326.3,A -85,B 0,C 180,E1 -15589.545,E2 -15589.545} C_VEL
LIN {X 0,Y 318.892,Z 314.079,A -85,B 0,C 180,E1 -15590.478,E2 -15590.478} C_VEL
LIN {X 0,Y 319.852,Z 301.346,A -85,B 0,C 180,E1 -15591.172,E2 -15591.172} C_VEL
LIN {X 0,Y 320.476,Z 288.235,A -85,B 0,C 180,E1 -15591.634,E2 -15591.634} C_VEL
LIN {X 0,Y 321.879,Z 225.387,A -85,B 0,C 180,E1 -15593.142,E2 -15593.142} C_VEL
LIN {X 0,Y 316.105,Z 183.703,A -85,B 0,C 180,E1 -15594.626,E2 -15594.626} C_VEL
LIN {X 0,Y 316.915,Z 176.939,A -85,B 0,C 180,E1 -15596.328,E2 -15596.328} C_VEL
LIN {X 0,Y 315.592,Z 168.616,A -85,B 0,C 180,E1 -15598.605,E2 -15598.605} C_VEL
LIN {X 0,Y 313.025,Z 156.817,A -85,B 0,C 180,E1 -15601.988,E2 -15601.988} C_VEL
LIN {X 0,Y 312.552,Z 154.554,A -85,B 0,C 180,E1 -15602.66,E2 -15602.66} C_VEL
LIN {X 0,Y 312.536,Z 154.556,A -85,B 0,C 180,E1 -15605.949,E2 -15605.949} C_VEL
LIN {X 0,Y 312.508,Z 154.555,A -85,B 0,C 180,E1 -15609.026,E2 -15609.026} C_VEL
LIN {X 0,Y 312.49,Z 154.559,A -85,B 0,C 180,E1 -15612.431,E2 -15612.431} C_VEL
LIN {X 0,Y 312.458,Z 154.564,A -85,B 0,C 180,E1 -15616.034,E2 -15616.034} C_VEL
LIN {X 0,Y 312.503,Z 154.559,A -85,B 0,C 180,E1 -15619.874,E2 -15619.874} C_VEL
LIN {X 0,Y 312.534,Z 154.553,A -85,B 0,C 180,E1 -15624.049,E2 -15624.049} C_VEL
LIN {X 0,Y 312.503,Z 154.559,A -85,B 0,C 180,E1 -15627.333,E2 -15627.333} C_VEL
LIN {X 0,Y 312.551,Z 154.552,A -85,B 0,C 180,E1 -15631.275,E2 -15631.275} C_VEL
LIN {X 0,Y 312.585,Z 154.546,A -85,B 0,C 180,E1 -15634.71,E2 -15634.71} C_VEL
LIN {X 0,Y 312.586,Z 154.548,A -85,B 0,C 180,E1 -15637.528,E2 -15637.528} C_VEL
LIN {X 0,Y 312.58,Z 154.547,A -85,B 0,C 180,E1 -15641.652,E2 -15641.652} C_VEL
LIN {X 0,Y 312.683,Z 154.534,A -85,B 0,C 180,E1 -15645.685,E2 -15645.685} C_VEL
LIN {X 0,Y 312.7,Z 154.531,A -85,B 0,C 180,E1 -15649.641,E2 -15649.641} C_VEL
LIN {X 0,Y 312.864,Z 154.509,A -85,B 0,C 180,E1 -15652.253,E2 -15652.253} C_VEL
LIN {X 0,Y 312.714,Z 154.533,A -85,B 0,C 180,E1 -15654.842,E2 -15654.842} C_VEL
LIN {X 0,Y 312.989,Z 154.499,A -85,B 0,C 180,E1 -15658.713,E2 -15658.713} C_VEL
LIN {X 0,Y 313.118,Z 154.478,A -85,B 0,C 180,E1 -15659.999,E2 -15659.999} C_VEL
LIN {X 0,Y 312.935,Z 154.503,A -85,B 0,C 180,E1 -15662.574,E2 -15662.574} C_VEL
LIN {X 0,Y 312.891,Z 154.509,A -85,B 0,C 180,E1 -15666.56,E2 -15666.56} C_VEL
LIN {X 0,Y 312.784,Z 154.522,A -85,B 0,C 180,E1 -15669.049,E2 -15669.049} C_VEL
LIN {X 0,Y 312.631,Z 154.538,A -85,B 0,C 180,E1 -15672.99,E2 -15672.99} C_VEL
LIN {X 0,Y 312.635,Z 154.537,A -85,B 0,C 180,E1 -15675.649,E2 -15675.649} C_VEL
LIN {X 0,Y 312.628,Z 154.54,A -85,B 0,C 180,E1 -15679.237,E2 -15679.237} C_VEL
LIN {X 0,Y 312.542,Z 154.551,A -85,B 0,C 180,E1 -15682.789,E2 -15682.789} C_VEL
LIN {X 0,Y 312.598,Z 154.542,A -85,B 0,C 180,E1 -15685.935,E2 -15685.935} C_VEL
LIN {X 0,Y 312.54,Z 154.551,A -85,B 0,C 180,E1 -15689.65,E2 -15689.65} C_VEL
LIN {X 0,Y 312.514,Z 154.554,A -85,B 0,C 180,E1 -15693.689,E2 -15693.689} C_VEL
LIN {X 0,Y 312.547,Z 154.548,A -85,B 0,C 180,E1 -15697.381,E2 -15697.381} C_VEL
LIN {X 0,Y 312.53,Z 154.552,A -85,B 0,C 180,E1 -15700.702,E2 -15700.702} C_VEL
LIN {X 0,Y 312.59,Z 154.546,A -85,B 0,C 180,E1 -15704.184,E2 -15704.184} C_VEL
LIN {X 0,Y 312.552,Z 154.554,A -85,B 0,C 180,E1 -15707.904,E2 -15707.904} C_VEL
LIN {X 0,Y 312.553,Z 154.553,A -85,B 0,C 180,E1 -15711.905,E2 -15711.905} C_VEL
LIN {X 0,Y 312.501,Z 154.56,A -85,B 0,C 180,E1 -15715.79,E2 -15715.79} C_VEL
LIN {X 0,Y 312.518,Z 154.554,A -85,B 0,C 180,E1 -15718.854,E2 -15718.854} C_VEL
LIN {X 0,Y 312.569,Z 154.55,A -85,B 0,C 180,E1 -15721.825,E2 -15721.825} C_VEL
LIN {X 0,Y 312.58,Z 154.546,A -85,B 0,C 180,E1 -15724.711,E2 -15724.711} C_VEL
LIN {X 0,Y 312.582,Z 154.551,A -85,B 0,C 180,E1 -15727.529,E2 -15727.529} C_VEL
LIN {X 0,Y 312.634,Z 154.542,A -85,B 0,C 180,E1 -15731.657,E2 -15731.657} C_VEL
LIN {X 0,Y 312.689,Z 154.535,A -85,B 0,C 180,E1 -15735.687,E2 -15735.687} C_VEL
LIN {X 0,Y 312.698,Z 154.533,A -85,B 0,C 180,E1 -15739.642,E2 -15739.642} C_VEL
LIN {X 0,Y 312.868,Z 154.51,A -85,B 0,C 180,E1 -15742.255,E2 -15742.255} C_VEL
LIN {X 0,Y 312.715,Z 154.532,A -85,B 0,C 180,E1 -15744.843,E2 -15744.843} C_VEL
LIN {X 0,Y 312.987,Z 154.498,A -85,B 0,C 180,E1 -15748.714,E2 -15748.714} C_VEL
LIN {X 0,Y 312.987,Z 154.498,A -85,B 0,C 180,E1 -15751.287,E2 -15751.287} C_VEL
LIN {X 0,Y 312.716,Z 154.532,A -85,B 0,C 180,E1 -15755.158,E2 -15755.158} C_VEL
LIN {X 0,Y 312.869,Z 154.51,A -85,B 0,C 180,E1 -15757.747,E2 -15757.747} C_VEL
LIN {X 0,Y 312.669,Z 154.538,A -85,B 0,C 180,E1 -15762.33,E2 -15762.33} C_VEL
LIN {X 0,Y 312.667,Z 154.665,A -85,B 0,C 180,E1 -15762.578,E2 -15762.578} C_VEL
LIN {X 0,Y 313.135,Z 156.797,A -85,B 0,C 180,E1 -15763.26,E2 -15763.26} C_VEL
LIN {X 0,Y 320.948,Z 178.629,A -85,B 0,C 180,E1 -15764.383,E2 -15764.383} C_VEL
LIN {X 0,Y 322.542,Z 184.232,A -85,B 0,C 180,E1 -15764.633,E2 -15764.633} C_VEL
LIN {X 0,Y 322.718,Z 189.809,A -85,B 0,C 180,E1 -15764.786,E2 -15764.786} C_VEL
LIN {X 0,Y 320.653,Z 265.001,A -85,B 0,C 180,E1 -15766.596,E2 -15766.596} C_VEL
LIN {X 0,Y 319.954,Z 278.23,A -85,B 0,C 180,E1 -15767.168,E2 -15767.168} C_VEL
LIN {X 0,Y 319.237,Z 290.505,A -85,B 0,C 180,E1 -15767.952,E2 -15767.952} C_VEL
LIN {X 0,Y 318.276,Z 302.618,A -85,B 0,C 180,E1 -15768.998,E2 -15768.998} C_VEL
LIN {X 0,Y 317.054,Z 314.087,A -85,B 0,C 180,E1 -15770.265,E2 -15770.265} C_VEL
LIN {X 0,Y 315.778,Z 324.871,A -85,B 0,C 180,E1 -15771.772,E2 -15771.772} C_VEL
LIN {X 0,Y 314.714,Z 333.717,A -85,B 0,C 180,E1 -15773.309,E2 -15773.309} C_VEL
LIN {X 0,Y 313.591,Z 342.565,A -85,B 0,C 180,E1 -15775.203,E2 -15775.203} C_VEL
LIN {X 0,Y 312.698,Z 349.59,A -85,B 0,C 180,E1 -15777.074,E2 -15777.074} C_VEL
LIN {X 0,Y 311.951,Z 355.627,A -85,B 0,C 180,E1 -15779.105,E2 -15779.105} C_VEL
LIN {X 0,Y 311.396,Z 360.579,A -85,B 0,C 180,E1 -15781.272,E2 -15781.272} C_VEL
LIN {X 0,Y 311.02,Z 363.959,A -85,B 0,C 180,E1 -15783.274,E2 -15783.274} C_VEL
LIN {X 0,Y 310.643,Z 366.463,A -85,B 0,C 180,E1 -15785.467,E2 -15785.467} C_VEL
LIN {X 0,Y 310.584,Z 367.777,A -85,B 0,C 180,E1 -15787.66,E2 -15787.66} C_VEL
LIN {X 0,Y 310.646,Z 367.956,A -85,B 0,C 180,E1 -15789.718,E2 -15789.718} C_VEL
LIN {X 0,Y 310.889,Z 367.135,A -85,B 0,C 180,E1 -15791.756,E2 -15791.756} C_VEL
LIN {X 0,Y 311.468,Z 364.581,A -85,B 0,C 180,E1 -15794.387,E2 -15794.387} C_VEL
LIN {X 0,Y 312.211,Z 360.583,A -85,B 0,C 180,E1 -15796.855,E2 -15796.855} C_VEL
LIN {X 0,Y 313.227,Z 355.558,A -85,B 0,C 180,E1 -15799.044,E2 -15799.044} C_VEL
LIN {X 0,Y 314.488,Z 348.795,A -85,B 0,C 180,E1 -15801.265,E2 -15801.265} C_VEL
LIN {X 0,Y 315.912,Z 341.229,A -85,B 0,C 180,E1 -15803.216,E2 -15803.216} C_VEL
LIN {X 0,Y 317.486,Z 332.563,A -85,B 0,C 180,E1 -15804.991,E2 -15804.991} C_VEL
LIN {X 0,Y 318.335,Z 327.483,A -85,B 0,C 180,E1 -15805.871,E2 -15805.871} C_VEL
LIN {X 0,Y 318.408,Z 323.193,A -85,B 0,C 180,E1 -15806.597,E2 -15806.597} C_VEL
LIN {X 0,Y 316.91,Z 316.069,A -85,B 0,C 180,E1 -15807.807,E2 -15807.807} C_VEL
LIN {X 0,Y 315.436,Z 308.523,A -85,B 0,C 180,E1 -15808.93,E2 -15808.93} C_VEL
LIN {X 0,Y 315.533,Z 303.485,A -85,B 0,C 180,E1 -15809.507,E2 -15809.507} C_VEL
LIN {X 0,Y 316.868,Z 291.567,A -85,B 0,C 180,E1 -15810.539,E2 -15810.539} C_VEL
LIN {X 0,Y 317.91,Z 278.571,A -85,B 0,C 180,E1 -15811.37,E2 -15811.37} C_VEL
LIN {X 0,Y 318.676,Z 266.17,A -85,B 0,C 180,E1 -15811.905,E2 -15811.905} C_VEL
LIN {X 0,Y 321.25,Z 190.641,A -85,B 0,C 180,E1 -15813.802,E2 -15813.802} C_VEL
LIN {X 0,Y 314.685,Z 175.248,A -85,B 0,C 180,E1 -15814.981,E2 -15814.981} C_VEL
LIN {X 0,Y 308.291,Z 162.672,A -85,B 0,C 180,E1 -15816.132,E2 -15816.132} C_VEL
LIN {X 0,Y 306.442,Z 159.11,A -85,B 0,C 180,E1 -15816.518,E2 -15816.518} C_VEL
LIN {X 0,Y 305.518,Z 155.433,A -85,B 0,C 180,E1 -15817.961,E2 -15817.961} C_VEL
LIN {X 0,Y 305.546,Z 155.426,A -85,B 0,C 180,E1 -15821.216,E2 -15821.216} C_VEL
LIN {X 0,Y 305.63,Z 155.419,A -85,B 0,C 180,E1 -15825.349,E2 -15825.349} C_VEL
LIN {X 0,Y 305.628,Z 155.414,A -85,B 0,C 180,E1 -15829.4,E2 -15829.4} C_VEL
LIN {X 0,Y 305.751,Z 155.4,A -85,B 0,C 180,E1 -15832.073,E2 -15832.073} C_VEL
LIN {X 0,Y 305.663,Z 155.411,A -85,B 0,C 180,E1 -15834.724,E2 -15834.724} C_VEL
LIN {X 0,Y 305.94,Z 155.369,A -85,B 0,C 180,E1 -15838.684,E2 -15838.684} C_VEL
LIN {X 0,Y 305.939,Z 155.376,A -85,B 0,C 180,E1 -15841.317,E2 -15841.317} C_VEL
LIN {X 0,Y 305.791,Z 155.383,A -85,B 0,C 180,E1 -15846.599,E2 -15846.599} C_VEL
LIN {X 0,Y 305.698,Z 155.405,A -85,B 0,C 180,E1 -15849.262,E2 -15849.262} C_VEL
LIN {X 0,Y 305.559,Z 155.422,A -85,B 0,C 180,E1 -15853.298,E2 -15853.298} C_VEL
LIN {X 0,Y 305.494,Z 155.423,A -85,B 0,C 180,E1 -15856.026,E2 -15856.026} C_VEL
LIN {X 0,Y 305.482,Z 155.423,A -85,B 0,C 180,E1 -15859.391,E2 -15859.391} C_VEL
LIN {X 0,Y 305.461,Z 155.429,A -85,B 0,C 180,E1 -15863.026,E2 -15863.026} C_VEL
LIN {X 0,Y 305.455,Z 155.435,A -85,B 0,C 180,E1 -15866.19,E2 -15866.19} C_VEL
LIN {X 0,Y 305.429,Z 155.437,A -85,B 0,C 180,E1 -15869.026,E2 -15869.026} C_VEL
LIN {X 0,Y 305.441,Z 155.431,A -85,B 0,C 180,E1 -15871.953,E2 -15871.953} C_VEL
LIN {X 0,Y 305.467,Z 155.428,A -85,B 0,C 180,E1 -15875.113,E2 -15875.113} C_VEL
LIN {X 0,Y 305.43,Z 155.434,A -85,B 0,C 180,E1 -15878.523,E2 -15878.523} C_VEL
LIN {X 0,Y 305.44,Z 155.441,A -85,B 0,C 180,E1 -15882.582,E2 -15882.582} C_VEL
LIN {X 0,Y 305.426,Z 155.441,A -85,B 0,C 180,E1 -15886.344,E2 -15886.344} C_VEL
LIN {X 0,Y 305.415,Z 155.446,A -85,B 0,C 180,E1 -15889.884,E2 -15889.884} C_VEL
LIN {X 0,Y 305.514,Z 155.552,A -85,B 0,C 180,E1 -15893.807,E2 -15893.807} C_VEL
LIN {X 0,Y 308.306,Z 166.242,A -85,B 0,C 180,E1 -15897.506,E2 -15897.506} C_VEL
LIN {X 0,Y 310.439,Z 175.605,A -85,B 0,C 180,E1 -15900.501,E2 -15900.501} C_VEL
LIN {X 0,Y 311.492,Z 181.277,A -85,B 0,C 180,E1 -15902.184,E2 -15902.184} C_VEL
LIN {X 0,Y 312.966,Z 185.885,A -85,B 0,C 180,E1 -15902.496,E2 -15902.496} C_VEL
LIN {X 0,Y 316.277,Z 201.78,A -85,B 0,C 180,E1 -15903.337,E2 -15903.337} C_VEL
LIN {X 0,Y 319.085,Z 219.507,A -85,B 0,C 180,E1 -15904.152,E2 -15904.152} C_VEL
LIN {X 0,Y 320.155,Z 228.527,A -85,B 0,C 180,E1 -15904.516,E2 -15904.516} C_VEL
LIN {X 0,Y 318.071,Z 291.094,A -85,B 0,C 180,E1 -15906.088,E2 -15906.088} C_VEL
LIN {X 0,Y 317.079,Z 304.474,A -85,B 0,C 180,E1 -15906.659,E2 -15906.659} C_VEL
